C05477=1141.444,-110.919,-44.146,178.630,6.023,149.486
C05478=1141.449,-111.169,-44.137,178.627,6.022,149.487
C05479=1141.455,-111.418,-44.129,178.625,6.021,149.487
C05480=1141.460,-111.668,-44.120,178.624,6.021,149.488
C05481=1141.465,-111.918,-44.111,178.621,6.021,149.488
C05482=1141.470,-112.168,-44.102,178.620,6.021,149.489
C05483=1141.476,-112.417,-44.094,178.618,6.020,149.489
C05484=1141.481,-112.667,-44.085,178.616,6.020,149.490
C05485=1141.487,-112.917,-44.077,178.614,6.019,149.490
C05486=1141.492,-113.167,-44.068,178.612,6.019,149.491
C05487=1141.498,-113.416,-44.059,178.610,6.019,149.491
C05488=1141.503,-113.667,-44.051,178.607,6.018,149.492
C05489=1141.508,-113.916,-44.042,178.606,6.018,149.492
C05490=1141.513,-114.166,-44.033,178.604,6.018,149.493
C05491=1141.519,-114.415,-44.025,178.602,6.018,149.493
C05492=1141.524,-114.665,-44.016,178.600,6.017,149.494
C05493=1141.530,-114.916,-44.008,178.598,6.016,149.494
C05494=1141.535,-115.166,-43.999,178.596,6.016,149.495
C05495=1141.541,-115.415,-43.990,178.594,6.015,149.495
C05496=1141.546,-115.665,-43.981,178.592,6.015,149.496
C05497=1141.551,-115.915,-43.973,178.590,6.015,149.496
C05498=1141.557,-116.164,-43.964,178.588,6.015,149.497
C05499=1141.562,-116.414,-43.956,178.586,6.014,149.497
C05500=1141.567,-116.664,-43.947,178.585,6.014,149.498
C05501=1141.573,-116.914,-43.938,178.582,6.013,149.498
C05502=1141.579,-117.164,-43.930,178.580,6.013,149.499
C05503=1141.584,-117.413,-43.921,178.579,6.013,149.499
C05504=1141.589,-117.663,-43.912,178.576,6.012,149.500
C05505=1141.595,-117.913,-43.904,178.574,6.012,149.500
C05506=1141.600,-118.163,-43.895,178.572,6.012,149.501
C05507=1141.605,-118.412,-43.887,178.571,6.012,149.501
C05508=1141.611,-118.662,-43.879,178.568,6.011,149.502
C05509=1141.616,-118.912,-43.870,178.567,6.011,149.502
C05510=1141.621,-119.162,-43.862,178.565,6.010,149.503
C05511=1141.627,-119.412,-43.854,178.563,6.010,149.503
C05512=1141.632,-119.662,-43.845,178.561,6.009,149.504
C05513=1141.637,-119.911,-43.836,178.559,6.009,149.504
C05514=1141.644,-120.161,-43.828,178.557,6.009,149.505
C05515=1141.649,-120.411,-43.819,178.555,6.008,149.505
C05516=1141.653,-120.661,-43.811,178.553,6.008,149.506
C05517=1141.659,-120.910,-43.803,178.551,6.007,149.506
C05518=1141.664,-121.160,-43.794,178.549,6.007,149.507
C05519=1141.670,-121.411,-43.786,178.547,6.007,149.507
C05520=1141.676,-121.660,-43.777,178.546,6.007,149.508
C05521=1141.681,-121.910,-43.769,178.543,6.006,149.508
C05522=1141.686,-122.160,-43.760,178.542,6.006,149.509
C05523=1141.691,-122.409,-43.752,178.540,6.005,149.509
C05524=1141.697,-122.659,-43.744,178.538,6.005,149.510
C05525=1141.702,-122.909,-43.735,178.536,6.004,149.510
C05526=1141.708,-123.158,-43.727,178.534,6.004,149.511
C05527=1141.713,-123.409,-43.719,178.532,6.004,149.511
C05528=1141.719,-123.658,-43.710,178.530,6.003,149.512
C05529=1141.724,-123.908,-43.703,178.528,6.003,149.512
C05530=1141.729,-124.158,-43.694,178.526,6.002,149.513
C05531=1141.735,-124.408,-43.686,178.524,6.002,149.513
C05532=1141.740,-124.658,-43.677,178.522,6.002,149.514
C05533=1141.746,-124.908,-43.669,178.521,6.002,149.514
C05534=1141.751,-125.157,-43.661,178.518,6.001,149.515
C05535=1141.756,-125.407,-43.653,178.517,6.001,149.515
C05536=1141.762,-125.657,-43.644,178.515,6.000,149.516
C05537=1141.767,-125.907,-43.636,178.513,6.000,149.516
C05538=1141.772,-126.157,-43.628,178.511,6.000,149.517
C05539=1141.778,-126.406,-43.620,178.509,6.000,149.517
C05540=1141.783,-126.656,-43.611,178.507,5.999,149.518
C05541=1141.789,-126.906,-43.603,178.505,5.999,149.518
C05542=1141.794,-127.156,-43.594,178.503,5.998,149.519
C05543=1141.799,-127.405,-43.587,178.502,5.998,149.519
C05544=1141.805,-127.655,-43.578,178.499,5.997,149.519
C05545=1141.810,-127.906,-43.570,178.498,5.997,149.520
C05546=1141.816,-128.155,-43.561,178.496,5.997,149.520
C05547=1141.821,-128.405,-43.554,178.494,5.997,149.521
C05548=1141.400,-128.416,-43.597,178.490,6.000,149.523
C05549=1141.395,-128.166,-43.605,178.492,6.001,149.522
C05550=1141.389,-127.916,-43.613,178.494,6.001,149.522
C05551=1141.384,-127.667,-43.622,178.496,6.001,149.521
C05552=1141.378,-127.417,-43.629,178.498,6.001,149.521
C05553=1141.373,-127.167,-43.638,178.500,6.002,149.520
C05554=1141.367,-126.917,-43.646,178.502,6.002,149.520
C05555=1141.363,-126.668,-43.654,178.504,6.003,149.519
C05556=1141.357,-126.417,-43.663,178.505,6.003,149.519
C05557=1141.351,-126.168,-43.671,178.508,6.004,149.518
C05558=1141.346,-125.918,-43.679,178.509,6.004,149.518
C05559=1141.340,-125.668,-43.688,178.511,6.004,149.517
C05560=1141.335,-125.418,-43.695,178.513,6.004,149.517
C05561=1141.330,-125.168,-43.704,178.515,6.005,149.516
C05562=1141.324,-124.919,-43.712,178.517,6.005,149.516
C05563=1141.319,-124.669,-43.721,178.519,6.006,149.515
C05564=1141.314,-124.419,-43.728,178.521,6.006,149.515
C05565=1141.308,-124.169,-43.737,178.523,6.006,149.514
C05566=1141.303,-123.919,-43.745,178.524,6.006,149.514
C05567=1141.297,-123.670,-43.754,178.527,6.007,149.513
C05568=1141.292,-123.419,-43.762,178.528,6.007,149.513
C05569=1141.286,-123.170,-43.771,178.530,6.008,149.513
C05570=1141.281,-122.920,-43.778,178.533,6.009,149.512
C05571=1141.276,-122.670,-43.787,178.534,6.008,149.512
C05572=1141.270,-122.421,-43.796,178.536,6.009,149.511
C05573=1141.265,-122.171,-43.804,178.538,6.009,149.511
C05574=1141.260,-121.921,-43.813,178.540,6.010,149.510
C05575=1141.254,-121.671,-43.821,178.542,6.010,149.510
C05576=1141.249,-121.421,-43.829,178.544,6.011,149.509
C05577=1141.244,-121.172,-43.838,178.546,6.011,149.509
C05578=1141.238,-120.922,-43.846,178.548,6.011,149.508
C05579=1141.233,-120.672,-43.854,178.549,6.011,149.508
C05580=1141.228,-120.422,-43.863,178.552,6.012,149.507
C05581=1141.222,-120.172,-43.871,178.553,6.012,149.507
C05582=1141.216,-119.922,-43.880,178.555,6.013,149.506
C05583=1141.212,-119.672,-43.888,178.557,6.013,149.506
C05584=1141.206,-119.423,-43.896,178.559,6.013,149.505
C05585=1141.201,-119.173,-43.905,178.561,6.014,149.505
C05586=1141.195,-118.923,-43.913,178.563,6.014,149.504
C05587=1141.189,-118.674,-43.922,178.565,6.015,149.504
C05588=1141.184,-118.424,-43.931,178.567,6.014,149.503
C05589=1141.179,-118.173,-43.939,178.569,6.015,149.503
C05590=1141.173,-117.924,-43.947,178.571,6.015,149.502
C05591=1141.168,-117.674,-43.956,178.573,6.016,149.502
C05592=1141.163,-117.425,-43.965,178.575,6.016,149.501
C05593=1141.157,-117.175,-43.973,178.577,6.017,149.501
C05594=1141.152,-116.925,-43.981,178.579,6.017,149.500
C05595=1141.147,-116.675,-43.990,178.581,6.017,149.500
C05596=1141.141,-116.426,-43.998,178.583,6.018,149.499
C05597=1141.136,-116.176,-44.007,178.585,6.018,149.499
C05598=1141.131,-115.926,-44.016,178.587,6.019,149.498
C05599=1141.125,-115.676,-44.025,178.588,6.019,149.498
C05600=1141.119,-115.426,-44.033,178.591,6.019,149.497
C05601=1141.114,-115.176,-44.041,178.592,6.019,149.497
C05602=1141.109,-114.927,-44.050,178.594,6.020,149.496
C05603=1141.103,-114.677,-44.059,178.597,6.021,149.496
C05604=1141.098,-114.427,-44.067,178.598,6.021,149.495
C05605=1141.093,-114.177,-44.076,178.600,6.022,149.495
C05606=1141.088,-113.927,-44.085,178.602,6.022,149.494
C05607=1141.082,-113.678,-44.093,178.605,6.022,149.494
C05608=1141.077,-113.428,-44.102,178.606,6.022,149.493
C05609=1141.071,-113.178,-44.110,178.608,6.023,149.493
C05610=1141.066,-112.928,-44.119,178.611,6.023,149.492
C05611=1141.060,-112.679,-44.128,178.612,6.023,149.492
C05612=1141.055,-112.429,-44.137,178.614,6.024,149.491
C05613=1141.050,-112.179,-44.146,178.616,6.024,149.491
C05614=1141.045,-111.929,-44.155,178.618,6.025,149.490
C05615=1141.039,-111.679,-44.162,178.620,6.025,149.490
C05616=1141.033,-111.430,-44.171,178.622,6.025,149.489
C05617=1141.028,-111.180,-44.180,178.624,6.026,149.489
C05618=1141.023,-110.930,-44.189,178.626,6.026,149.488
C05619=1141.018,-110.680,-44.198,178.628,6.027,149.488
C05620=1141.012,-110.431,-44.207,178.630,6.027,149.487
C05621=1141.006,-110.181,-44.216,178.632,6.027,149.487
C05622=1141.001,-109.931,-44.225,178.634,6.027,149.486
C05623=1140.996,-109.680,-44.233,178.636,6.028,149.486
C05624=1140.990,-109.431,-44.242,178.638,6.029,149.485
C05625=1140.985,-109.181,-44.251,178.640,6.029,149.485
C05626=1140.980,-108.932,-44.259,178.642,6.029,149.484
C05627=1140.974,-108.682,-44.268,178.644,6.029,149.484
C05628=1140.969,-108.432,-44.277,178.646,6.030,149.483
C05629=1140.963,-108.183,-44.286,178.648,6.031,149.483
C05630=1140.958,-107.933,-44.295,178.650,6.031,149.482
C05631=1140.953,-107.683,-44.304,178.652,6.031,149.481
C05632=1140.948,-107.433,-44.312,178.654,6.031,149.481
C05633=1140.942,-107.183,-44.322,178.656,6.032,149.480
C05634=1140.937,-106.933,-44.331,178.658,6.033,149.480
C05635=1140.931,-106.684,-44.339,178.660,6.033,149.479
C05636=1140.926,-106.434,-44.348,178.662,6.033,149.479
C05637=1140.921,-106.184,-44.357,178.664,6.033,149.479
C05638=1140.916,-105.934,-44.366,178.666,6.034,149.478
C05639=1140.910,-105.685,-44.375,178.668,6.035,149.478
C05640=1140.905,-105.435,-44.384,178.670,6.035,149.477
C05641=1140.899,-105.185,-44.393,178.672,6.035,149.476
C05642=1140.894,-104.935,-44.402,178.674,6.035,149.476
C05643=1140.888,-104.686,-44.411,178.676,6.036,149.475
C05644=1140.883,-104.436,-44.420,178.678,6.037,149.475
C05645=1140.878,-104.186,-44.429,178.680,6.037,149.474
C05646=1140.873,-103.936,-44.437,178.682,6.037,149.474
C05647=1140.867,-103.686,-44.447,178.684,6.037,149.473
C05648=1140.862,-103.436,-44.456,178.686,6.038,149.473
C05649=1140.856,-103.165,-44.466,178.689,6.038,149.472
C05650=1140.850,-102.892,-44.475,178.691,6.039,149.472
C05651=1140.844,-102.620,-44.485,178.692,6.039,149.471
C05652=1140.839,-102.348,-44.495,178.695,6.039,149.471
C05653=1140.833,-102.098,-44.504,178.697,6.040,149.470
C05654=1140.828,-101.848,-44.513,178.699,6.040,149.470
C05655=1140.822,-101.598,-44.522,178.701,6.041,149.469
C05656=1140.817,-101.348,-44.531,178.703,6.042,149.469
C05657=1140.811,-101.099,-44.540,178.705,6.042,149.468
C05658=1140.807,-100.850,-44.549,178.707,6.042,149.468
C05659=1140.801,-100.600,-44.559,178.710,6.043,149.467
C05660=1140.796,-100.350,-44.568,178.711,6.043,149.466
C05661=1140.790,-100.100,-44.577,178.713,6.043,149.466
C05662=1140.785,-99.850,-44.585,178.715,6.043,149.465
C05663=1140.779,-99.600,-44.595,178.717,6.044,149.465
C05664=1140.774,-99.351,-44.605,178.719,6.045,149.464
C05665=1140.769,-99.101,-44.613,178.721,6.045,149.464
C05666=1140.763,-98.851,-44.623,178.724,6.045,149.463
C05667=1140.758,-98.601,-44.632,178.726,6.046,149.463
C05668=1140.753,-98.351,-44.641,178.728,6.046,149.462
C05669=1140.747,-98.102,-44.649,178.730,6.047,149.462
C05670=1140.742,-97.852,-44.660,178.732,6.047,149.461
C05671=1140.737,-97.602,-44.668,178.734,6.047,149.461
C05672=1140.731,-97.352,-44.677,178.736,6.048,149.460
C05673=1140.725,-97.102,-44.687,178.738,6.048,149.460
C05674=1140.721,-96.853,-44.696,178.740,6.049,149.459
C05675=1140.715,-96.603,-44.705,178.742,6.049,149.459
C05676=1140.710,-96.353,-44.715,178.744,6.049,149.458
C05677=1140.704,-96.103,-44.724,178.746,6.050,149.458
C05678=1140.699,-95.854,-44.733,178.748,6.051,149.457
C05679=1140.694,-95.604,-44.743,178.750,6.051,149.457
C05680=1140.688,-95.354,-44.752,178.752,6.051,149.456
C05681=1140.683,-95.104,-44.761,178.755,6.052,149.456
C05682=1140.678,-94.855,-44.771,178.756,6.052,149.455
C05683=1140.672,-94.605,-44.780,178.758,6.053,149.455
C05684=1140.667,-94.355,-44.789,178.761,6.053,149.454
C05685=1140.662,-94.105,-44.799,178.762,6.053,149.454
C05686=1140.657,-93.855,-44.808,178.765,6.054,149.453
C05687=1140.651,-93.606,-44.817,178.767,6.054,149.452
C05688=1140.646,-93.356,-44.827,178.769,6.054,149.452
C05689=1140.641,-93.106,-44.836,178.771,6.055,149.451
C05690=1140.635,-92.856,-44.845,178.773,6.056,149.451
C05691=1140.630,-92.607,-44.855,178.775,6.056,149.450
C05692=1140.625,-92.357,-44.864,178.777,6.056,149.450
C05693=1140.619,-92.107,-44.873,178.780,6.057,149.449
C05694=1140.614,-91.858,-44.883,178.781,6.057,149.449
C05695=1140.608,-91.607,-44.892,178.783,6.058,149.448
C05696=1140.603,-91.358,-44.901,178.786,6.058,149.448
C05697=1140.598,-91.108,-44.911,178.787,6.058,149.447
C05698=1140.592,-90.858,-44.920,178.790,6.059,149.447
C05699=1140.587,-90.609,-44.930,178.792,6.060,149.446
C05700=1140.581,-90.359,-44.939,178.794,6.060,149.446
C05701=1140.576,-90.109,-44.948,178.796,6.060,149.445
C05702=1140.571,-89.859,-44.959,178.798,6.061,149.445
C05703=1140.565,-89.610,-44.967,178.800,6.061,149.444
C05704=1140.560,-89.360,-44.978,178.802,6.061,149.443
C05705=1140.555,-89.110,-44.987,178.804,6.062,149.443
C05706=1140.550,-88.860,-44.997,178.806,6.062,149.443
C05707=1140.544,-88.610,-45.006,178.808,6.063,149.442
C05708=1140.540,-88.361,-45.016,178.810,6.064,149.442
C05709=1140.534,-88.111,-45.025,178.813,6.064,149.441
C05710=1140.529,-87.861,-45.034,178.815,6.064,149.440
C05711=1140.523,-87.611,-45.044,178.817,6.065,149.440
C05712=1140.518,-87.361,-45.053,178.819,6.065,149.439
C05713=1140.512,-87.112,-45.063,178.821,6.065,149.439
C05714=1140.507,-86.862,-45.072,178.823,6.066,149.438
C05715=1140.501,-86.612,-45.082,178.826,6.067,149.438
C05716=1140.496,-86.363,-45.091,178.827,6.067,149.437
C05717=1140.491,-86.113,-45.102,178.829,6.067,149.437
C05718=1140.486,-85.863,-45.112,178.831,6.068,149.436
C05719=1140.480,-85.613,-45.121,178.834,6.068,149.436
C05720=1140.476,-85.364,-45.131,178.836,6.068,149.435
C05721=1140.470,-85.114,-45.140,178.838,6.069,149.435
C05722=1140.465,-84.864,-45.150,178.840,6.070,149.434
C05723=1140.459,-84.614,-45.159,178.842,6.070,149.434
C05724=1140.453,-84.365,-45.169,178.844,6.070,149.433
C05725=1140.448,-84.115,-45.178,178.847,6.071,149.432
C05726=1140.443,-83.865,-45.189,178.849,6.072,149.432
C05727=1140.438,-83.615,-45.199,178.850,6.072,149.431
C05728=1140.432,-83.365,-45.208,178.853,6.072,149.431
C05729=1140.428,-83.116,-45.218,178.855,6.073,149.430
C05730=1140.422,-82.866,-45.227,178.857,6.073,149.430
C05731=1140.416,-82.616,-45.237,178.859,6.074,149.429
C05732=1140.411,-82.367,-45.247,178.861,6.074,149.429
C05733=1140.406,-82.116,-45.257,178.863,6.075,149.428
C05734=1140.401,-81.867,-45.266,178.866,6.075,149.428
C05735=1140.395,-81.617,-45.277,178.868,6.075,149.427
C05736=1140.390,-81.367,-45.286,178.870,6.076,149.427
C05737=1140.385,-81.118,-45.296,178.871,6.076,149.426
C05738=1140.379,-80.868,-45.306,178.874,6.077,149.425
C05739=1140.375,-80.618,-45.315,178.876,6.077,149.425
C05740=1140.369,-80.368,-45.325,178.879,6.078,149.424
C05741=1140.363,-80.119,-45.336,178.880,6.078,149.424
C05742=1140.358,-79.869,-45.345,178.882,6.079,149.424
C05743=1140.353,-79.619,-45.355,178.885,6.079,149.423
C05744=1140.347,-79.370,-45.365,178.887,6.080,149.422
C05745=1140.343,-79.120,-45.375,178.889,6.080,149.422
C05746=1140.337,-78.870,-45.384,178.891,6.081,149.421
C05747=1140.331,-78.620,-45.395,178.894,6.081,149.421
C05748=1140.326,-78.371,-45.404,178.896,6.082,149.420
C05749=1140.320,-78.121,-45.414,178.897,6.082,149.420
C05750=1140.315,-77.871,-45.424,178.900,6.083,149.419
C05751=1140.310,-77.621,-45.435,178.902,6.083,149.419
C05752=1140.305,-77.372,-45.444,178.905,6.084,149.418
C05753=1140.299,-77.100,-45.455,178.906,6.084,149.418
C05754=1140.293,-76.829,-45.466,178.909,6.084,149.417
C05755=1140.287,-76.557,-45.477,178.911,6.085,149.416
C05756=1140.282,-76.285,-45.487,178.913,6.086,149.416
C05757=1140.276,-76.036,-45.498,178.916,6.086,149.415
C05758=1140.271,-75.787,-45.507,178.918,6.087,149.415
C05759=1140.266,-75.536,-45.518,178.920,6.087,149.414
C05760=1140.260,-75.287,-45.528,178.922,6.087,149.414
C05761=1140.255,-75.037,-45.537,178.925,6.088,149.413
C05762=1140.250,-74.787,-45.547,178.927,6.089,149.412
C05763=1140.244,-74.538,-45.557,178.928,6.088,149.412
C05764=1140.239,-74.288,-45.568,178.930,6.089,149.412
C05765=1140.234,-74.038,-45.578,178.933,6.090,149.411
C05766=1140.228,-73.789,-45.588,178.935,6.090,149.410
C05767=1140.223,-73.538,-45.597,178.938,6.091,149.410
C05768=1140.218,-73.288,-45.608,178.939,6.091,149.409
C05769=1140.212,-73.039,-45.618,178.942,6.092,149.409
C05770=1140.207,-72.789,-45.628,178.944,6.092,149.408
C05771=1140.202,-72.539,-45.638,178.946,6.093,149.408
C05772=1140.197,-72.290,-45.648,178.948,6.093,149.407
C05773=1140.191,-72.040,-45.659,178.950,6.093,149.407
C05774=1140.185,-71.791,-45.669,178.953,6.094,149.406
C05775=1140.181,-71.541,-45.679,178.955,6.095,149.406
C05776=1140.175,-71.291,-45.689,178.956,6.095,149.405
C05777=1140.170,-71.042,-45.699,178.959,6.095,149.404
C05778=1140.165,-70.792,-45.710,178.961,6.096,149.404
C05779=1140.159,-70.542,-45.720,178.963,6.097,149.403
C05780=1140.154,-70.292,-45.729,178.966,6.098,149.403
C05781=1140.149,-70.042,-45.740,178.968,6.097,149.402
C05782=1140.143,-69.792,-45.750,178.970,6.098,149.402
C05783=1140.138,-69.543,-45.760,178.972,6.099,149.401
C05784=1140.133,-69.293,-45.770,178.974,6.099,149.401
C05785=1140.127,-69.043,-45.781,178.977,6.100,149.400
C05786=1140.122,-68.794,-45.791,178.979,6.100,149.400
C05787=1140.117,-68.543,-45.801,178.981,6.101,149.399
C05788=1140.111,-68.294,-45.812,178.983,6.101,149.399
C05789=1140.106,-68.045,-45.822,178.986,6.102,149.398
C05790=1140.101,-67.795,-45.833,178.988,6.102,149.397
C05791=1140.095,-67.545,-45.843,178.989,6.102,149.397
C05792=1140.091,-67.296,-45.853,178.992,6.103,149.396
C05793=1140.086,-67.046,-45.863,178.994,6.104,149.396
C05794=1140.080,-66.796,-45.874,178.996,6.104,149.395
C05795=1140.074,-66.546,-45.884,178.999,6.105,149.395
C05796=1140.069,-66.296,-45.894,179.001,6.105,149.394
C05797=1140.064,-66.047,-45.905,179.003,6.106,149.394
C05798=1140.059,-65.796,-45.915,179.005,6.106,149.393
C05799=1140.053,-65.547,-45.925,179.007,6.107,149.393
C05800=1140.048,-65.297,-45.936,179.010,6.107,149.392
C05801=1140.043,-65.047,-45.946,179.012,6.107,149.391
C05802=1140.037,-64.798,-45.957,179.014,6.108,149.391
C05803=1140.032,-64.548,-45.968,179.016,6.109,149.390
C05804=1140.027,-64.298,-45.978,179.019,6.109,149.390
C05805=1140.021,-64.049,-45.988,179.021,6.110,149.389
C05806=1140.016,-63.799,-45.999,179.023,6.111,149.389
C05807=1140.010,-63.549,-46.009,179.025,6.110,149.388
C05808=1140.006,-63.299,-46.020,179.027,6.111,149.388
C05809=1140.000,-63.050,-46.030,179.029,6.112,149.387
C05810=1139.995,-62.800,-46.041,179.032,6.113,149.387
C05811=1139.990,-62.550,-46.051,179.034,6.113,149.386
C05812=1139.984,-62.301,-46.061,179.036,6.113,149.385
C05813=1139.979,-62.051,-46.073,179.038,6.114,149.385
C05814=1139.974,-61.801,-46.083,179.041,6.114,149.384
C05815=1139.969,-61.551,-46.093,179.043,6.115,149.384
C05816=1139.963,-61.302,-46.104,179.045,6.116,149.383
C05817=1139.958,-61.051,-46.114,179.047,6.117,149.383
C05818=1139.953,-60.802,-46.125,179.049,6.116,149.382
C05819=1139.947,-60.553,-46.135,179.052,6.117,149.382
C05820=1139.942,-60.303,-46.146,179.054,6.118,149.381
C05821=1139.937,-60.053,-46.156,179.056,6.118,149.380
C05822=1139.932,-59.803,-46.167,179.059,6.119,149.380
C05823=1139.926,-59.554,-46.178,179.061,6.120,149.380
C05824=1139.921,-59.304,-46.188,179.063,6.120,149.379
C05825=1139.916,-59.055,-46.199,179.065,6.120,149.378
C05826=1139.911,-58.805,-46.210,179.067,6.121,149.378
C05827=1139.905,-58.555,-46.220,179.069,6.122,149.377
C05828=1139.901,-58.305,-46.231,179.072,6.122,149.377
C05829=1139.895,-58.056,-46.241,179.074,6.123,149.376
C05830=1139.890,-57.806,-46.252,179.077,6.123,149.376
C05831=1139.885,-57.557,-46.263,179.079,6.124,149.375
C05832=1139.879,-57.306,-46.274,179.081,6.124,149.375
C05833=1139.874,-57.057,-46.284,179.083,6.125,149.374
C05834=1139.869,-56.807,-46.296,179.085,6.125,149.374
C05835=1139.863,-56.557,-46.306,179.088,6.126,149.373
C05836=1139.858,-56.307,-46.316,179.090,6.127,149.372
C05837=1139.853,-56.058,-46.327,179.092,6.127,149.372
C05838=1139.848,-55.808,-46.338,179.095,6.128,149.371
C05839=1139.843,-55.559,-46.349,179.096,6.128,149.371
C05840=1139.837,-55.308,-46.360,179.099,6.128,149.370
C05841=1139.831,-55.059,-46.370,179.101,6.129,149.370
C05842=1139.827,-54.809,-46.381,179.104,6.130,149.369
C05843=1139.822,-54.559,-46.392,179.106,6.130,149.369
C05844=1139.816,-54.310,-46.403,179.108,6.131,149.368
C05845=1139.811,-54.060,-46.414,179.111,6.132,149.367
C05846=1139.805,-53.811,-46.425,179.113,6.132,149.367
C05847=1139.800,-53.560,-46.436,179.114,6.132,149.366
C05848=1139.795,-53.311,-46.447,179.117,6.133,149.366
C05849=1139.790,-53.061,-46.457,179.119,6.133,149.365
C05850=1139.784,-52.812,-46.467,179.121,6.134,149.365
C05851=1139.779,-52.562,-46.479,179.124,6.135,149.364
C05852=1139.774,-52.311,-46.490,179.126,6.135,149.364
C05853=1139.769,-52.063,-46.501,179.128,6.136,149.363
C05854=1139.764,-51.812,-46.511,179.131,6.137,149.363
C05855=1139.758,-51.563,-46.523,179.133,6.137,149.362
C05856=1139.753,-51.313,-46.534,179.135,6.137,149.361
C05857=1139.747,-51.042,-46.546,179.138,6.138,149.361
C05858=1139.742,-50.772,-46.557,179.140,6.138,149.360
C05859=1139.736,-50.501,-46.569,179.143,6.140,149.360
C05860=1139.730,-50.230,-46.581,179.145,6.140,149.359
C05861=1139.725,-49.981,-46.592,179.147,6.140,149.359
C05862=1139.720,-49.731,-46.603,179.149,6.141,149.358
C05863=1139.714,-49.482,-46.614,179.152,6.142,149.357
C05864=1139.709,-49.231,-46.625,179.154,6.142,149.357
C05865=1139.704,-48.982,-46.636,179.157,6.143,149.356
C05866=1139.698,-48.732,-46.648,179.159,6.144,149.356
C05867=1139.693,-48.482,-46.658,179.161,6.144,149.355
C05868=1139.688,-48.233,-46.669,179.164,6.145,149.355
C05869=1139.682,-47.983,-46.681,179.166,6.145,149.354
C05870=1139.678,-47.733,-46.692,179.168,6.146,149.354
C05871=1139.672,-47.484,-46.703,179.171,6.147,149.353
C05872=1139.667,-47.234,-46.713,179.172,6.147,149.352
C05873=1139.662,-46.984,-46.725,179.174,6.147,149.352
C05874=1139.657,-46.735,-46.736,179.177,6.148,149.352
C05875=1139.651,-46.484,-46.747,179.179,6.149,149.351
C05876=1139.646,-46.235,-46.759,179.181,6.149,149.350
C05877=1139.641,-45.986,-46.770,179.184,6.150,149.350
C05878=1139.635,-45.735,-46.781,179.186,6.151,149.349
C05879=1139.630,-45.486,-46.792,179.188,6.151,149.349
C05880=1139.625,-45.237,-46.803,179.191,6.152,149.348
C05881=1139.620,-44.987,-46.815,179.193,6.152,149.347
C05882=1139.615,-44.737,-46.825,179.196,6.153,149.347
C05883=1139.609,-44.488,-46.836,179.198,6.154,149.347
C05884=1139.604,-44.238,-46.848,179.200,6.154,149.346
C05885=1139.599,-43.988,-46.859,179.203,6.155,149.345
C05886=1139.593,-43.738,-46.870,179.204,6.155,149.345
C05887=1139.588,-43.489,-46.882,179.207,6.156,149.344
C05888=1139.583,-43.239,-46.893,179.209,6.156,149.344
C05889=1139.578,-42.989,-46.905,179.211,6.157,149.343
C05890=1139.573,-42.740,-46.915,179.214,6.158,149.343
C05891=1139.567,-42.490,-46.927,179.216,6.158,149.342
C05892=1139.562,-42.240,-46.938,179.218,6.159,149.342
C05893=1139.556,-41.991,-46.950,179.221,6.160,149.341
C05894=1139.552,-41.741,-46.961,179.223,6.160,149.340
C05895=1139.546,-41.491,-46.972,179.225,6.161,149.340
C05896=1139.541,-41.241,-46.983,179.228,6.161,149.339
C05897=1139.535,-40.992,-46.995,179.230,6.162,149.339
C05898=1139.531,-40.742,-47.006,179.232,6.163,149.338
C05899=1139.526,-40.493,-47.017,179.235,6.163,149.338
C05900=1139.520,-40.243,-47.029,179.237,6.164,149.337
C05901=1139.515,-39.994,-47.040,179.239,6.165,149.337
C05902=1139.509,-39.743,-47.051,179.242,6.165,149.336
C05903=1139.505,-39.493,-47.063,179.244,6.166,149.335
C05904=1139.499,-39.244,-47.075,179.246,6.167,149.335
C05905=1139.493,-38.994,-47.086,179.249,6.167,149.334
C05906=1139.489,-38.745,-47.097,179.251,6.167,149.334
C05907=1139.483,-38.495,-47.109,179.253,6.168,149.333
C05908=1139.478,-38.245,-47.121,179.256,6.169,149.333
C05909=1139.473,-37.995,-47.133,179.258,6.169,149.332
C05910=1139.468,-37.746,-47.143,179.260,6.170,149.332
C05911=1139.462,-37.496,-47.155,179.263,6.170,149.331
C05912=1139.458,-37.247,-47.167,179.265,6.171,149.330
C05913=1139.452,-36.997,-47.178,179.267,6.172,149.330
C05914=1139.447,-36.747,-47.190,179.270,6.172,149.329
C05915=1139.441,-36.498,-47.201,179.272,6.173,149.329
C05916=1139.436,-36.248,-47.213,179.274,6.174,149.328
C05917=1139.431,-35.998,-47.224,179.277,6.174,149.328
C05918=1139.426,-35.748,-47.236,179.279,6.175,149.327
C05919=1139.421,-35.499,-47.248,179.281,6.176,149.326
C05920=1139.415,-35.250,-47.259,179.284,6.176,149.326
C05921=1139.410,-35.000,-47.271,179.286,6.177,149.326
C05922=1139.405,-34.750,-47.282,179.289,6.178,149.325
C05923=1139.400,-34.500,-47.294,179.291,6.178,149.324
C05924=1139.395,-34.250,-47.306,179.293,6.179,149.324
C05925=1139.390,-34.000,-47.317,179.296,6.180,149.323
C05926=1139.383,-33.751,-47.329,179.298,6.180,149.323
C05927=1139.379,-33.502,-47.340,179.300,6.181,149.322
C05928=1139.373,-33.252,-47.352,179.303,6.181,149.322
C05929=1139.368,-33.002,-47.364,179.305,6.182,149.321
C05930=1139.363,-32.752,-47.375,179.307,6.183,149.321
C05931=1139.358,-32.502,-47.387,179.310,6.183,149.320
C05932=1139.353,-32.253,-47.400,179.312,6.184,149.319
C05933=1139.347,-32.004,-47.411,179.314,6.185,149.319
C05934=1139.342,-31.754,-47.423,179.317,6.185,149.318
C05935=1139.337,-31.504,-47.434,179.319,6.186,149.318
C05936=1139.332,-31.254,-47.446,179.321,6.187,149.317
C05937=1139.326,-31.004,-47.458,179.324,6.187,149.317
C05938=1139.321,-30.755,-47.470,179.326,6.188,149.316
C05939=1139.317,-30.506,-47.482,179.328,6.189,149.316
C05940=1139.311,-30.256,-47.493,179.331,6.189,149.315
C05941=1139.306,-30.006,-47.505,179.333,6.190,149.314
C05942=1139.300,-29.756,-47.517,179.336,6.191,149.314
C05943=1139.295,-29.507,-47.528,179.338,6.191,149.313
C05944=1139.290,-29.258,-47.541,179.340,6.192,149.313
C05945=1139.284,-29.008,-47.553,179.343,6.193,149.312
C05946=1139.280,-28.758,-47.564,179.345,6.193,149.312
C05947=1139.274,-28.508,-47.576,179.347,6.194,149.311
C05948=1139.269,-28.259,-47.588,179.350,6.195,149.310
C05949=1139.264,-28.009,-47.600,179.352,6.195,149.310
C05950=1139.259,-27.759,-47.612,179.354,6.196,149.310
C05951=1139.254,-27.509,-47.623,179.357,6.197,149.309
C05952=1139.249,-27.260,-47.636,179.359,6.198,149.308
C05953=1139.243,-27.010,-47.648,179.362,6.199,149.308
C05954=1139.238,-26.760,-47.660,179.364,6.199,149.307
C05955=1139.233,-26.510,-47.671,179.366,6.200,149.307
C05956=1139.228,-26.261,-47.684,179.369,6.200,149.306
C05957=1139.222,-26.011,-47.696,179.371,6.201,149.306
C05958=1139.217,-25.761,-47.707,179.374,6.202,149.305
C05959=1139.212,-25.512,-47.720,179.376,6.202,149.304
C05960=1139.207,-25.262,-47.731,179.378,6.203,149.304
C05961=1139.201,-24.992,-47.745,179.381,6.204,149.303
C05962=1139.195,-24.722,-47.758,179.383,6.204,149.303
C05963=1139.190,-24.452,-47.770,179.386,6.206,149.302
C05964=1139.184,-24.183,-47.784,179.389,6.206,149.302
C05965=1139.179,-23.933,-47.796,179.391,6.207,149.301
C05966=1139.173,-23.683,-47.808,179.394,6.208,149.300
C05967=1139.168,-23.433,-47.820,179.396,6.208,149.300
C05968=1139.163,-23.183,-47.832,179.398,6.209,149.299
C05969=1139.159,-22.934,-47.844,179.401,6.210,149.299
C05970=1139.153,-22.684,-47.856,179.403,6.210,149.298
C05971=1139.148,-22.435,-47.868,179.405,6.211,149.298
C05972=1139.143,-22.185,-47.880,179.408,6.212,149.297
C05973=1139.137,-21.935,-47.892,179.410,6.212,149.297
C05974=1139.132,-21.686,-47.905,179.412,6.213,149.296
C05975=1139.127,-21.436,-47.917,179.415,6.214,149.295
C05976=1139.121,-21.187,-47.929,179.418,6.215,149.295
C05977=1139.117,-20.936,-47.942,179.420,6.216,149.294
C05978=1139.111,-20.687,-47.954,179.422,6.216,149.294
C05979=1139.106,-20.437,-47.966,179.425,6.217,149.293
C05980=1139.101,-20.187,-47.979,179.427,6.218,149.293
C05981=1139.096,-19.938,-47.991,179.429,6.218,149.292
C05982=1139.091,-19.689,-48.003,179.432,6.219,149.291
C05983=1139.086,-19.439,-48.015,179.434,6.220,149.291
C05984=1139.081,-19.189,-48.027,179.436,6.220,149.291
C05985=1139.075,-18.939,-48.039,179.439,6.221,149.290
C05986=1139.070,-18.690,-48.052,179.441,6.222,149.289
C05987=1139.065,-18.441,-48.064,179.444,6.222,149.289
C05988=1139.059,-18.191,-48.076,179.447,6.224,149.288
C05989=1139.054,-17.941,-48.089,179.449,6.224,149.288
C05990=1139.049,-17.692,-48.101,179.451,6.225,149.287
C05991=1139.044,-17.442,-48.114,179.454,6.226,149.287
C05992=1139.039,-17.192,-48.125,179.456,6.226,149.286
C05993=1139.034,-16.942,-48.138,179.458,6.227,149.285
C05994=1139.029,-16.693,-48.151,179.461,6.228,149.285
C05995=1139.023,-16.443,-48.163,179.463,6.228,149.284
C05996=1139.018,-16.194,-48.175,179.465,6.229,149.284
C05997=1139.013,-15.944,-48.188,179.468,6.230,149.283
C05998=1139.007,-15.694,-48.200,179.471,6.231,149.283
C05999=1139.002,-15.444,-48.213,179.473,6.232,149.282
C06000=1138.997,-15.195,-48.226,179.475,6.232,149.282
C06001=1138.992,-14.945,-48.238,179.478,6.233,149.281
C06002=1138.987,-14.696,-48.250,179.480,6.234,149.281
C06003=1138.982,-14.446,-48.263,179.482,6.234,149.280
C06004=1138.976,-14.196,-48.275,179.485,6.235,149.279
C06005=1138.971,-13.947,-48.287,179.487,6.236,149.279
C06006=1138.966,-13.697,-48.300,179.490,6.236,149.278
C06007=1138.961,-13.448,-48.313,179.493,6.238,149.278
C06008=1138.956,-13.198,-48.325,179.495,6.238,149.277
C06009=1138.951,-12.948,-48.337,179.497,6.239,149.277
C06010=1138.945,-12.699,-48.351,179.500,6.240,149.276
C06011=1138.940,-12.449,-48.364,179.502,6.240,149.276
C06012=1138.935,-12.199,-48.375,179.504,6.241,149.275
C06013=1138.930,-11.949,-48.388,179.507,6.242,149.274
C06014=1138.925,-11.700,-48.401,179.509,6.242,149.274
C06015=1138.920,-11.451,-48.413,179.512,6.244,149.273
C06016=1138.914,-11.202,-48.426,179.514,6.244,149.273
C06017=1138.910,-10.951,-48.438,179.517,6.245,149.272
C06018=1138.904,-10.701,-48.451,179.519,6.246,149.272
C06019=1138.899,-10.452,-48.464,179.521,6.246,149.271
C06020=1138.894,-10.203,-48.476,179.524,6.247,149.271
C06021=1138.889,-9.953,-48.489,179.526,6.248,149.270
C06022=1138.884,-9.703,-48.502,179.529,6.249,149.270
C06023=1138.878,-9.453,-48.515,179.532,6.250,149.269
C06024=1138.873,-9.204,-48.527,179.534,6.251,149.268
C06025=1138.868,-8.954,-48.540,179.536,6.251,149.268
C06026=1138.863,-8.704,-48.553,179.539,6.252,149.267
C06027=1138.858,-8.455,-48.565,179.541,6.253,149.267
C06028=1138.852,-8.205,-48.578,179.543,6.253,149.266
C06029=1138.847,-7.955,-48.591,179.546,6.255,149.266
C06030=1138.842,-7.706,-48.604,179.548,6.255,149.265
C06031=1138.837,-7.457,-48.617,179.551,6.256,149.264
C06032=1138.831,-7.207,-48.630,179.553,6.257,149.264
C06033=1138.827,-6.957,-48.643,179.556,6.257,149.263
C06034=1138.822,-6.708,-48.655,179.558,6.258,149.263
C06035=1138.817,-6.458,-48.668,179.561,6.259,149.262
C06036=1138.811,-6.209,-48.681,179.563,6.260,149.262
C06037=1138.806,-5.959,-48.694,179.566,6.261,149.261
C06038=1138.801,-5.710,-48.707,179.568,6.261,149.261
C06039=1138.796,-5.460,-48.719,179.570,6.262,149.260
C06040=1138.791,-5.210,-48.733,179.573,6.263,149.260
C06041=1138.786,-4.961,-48.746,179.576,6.264,149.259
C06042=1138.780,-4.711,-48.758,179.578,6.265,149.258
C06043=1138.775,-4.461,-48.772,179.580,6.265,149.258
C06044=1138.770,-4.212,-48.784,179.583,6.266,149.257
C06045=1138.765,-3.962,-48.797,179.585,6.267,149.257
C06046=1138.760,-3.712,-48.810,179.588,6.268,149.256
C06047=1138.755,-3.463,-48.823,179.591,6.269,149.256
C06048=1138.749,-3.213,-48.836,179.593,6.269,149.255
C06049=1138.744,-2.963,-48.849,179.595,6.270,149.254
C06050=1138.739,-2.714,-48.862,179.598,6.271,149.254
C06051=1138.734,-2.464,-48.874,179.600,6.272,149.254
C06052=1138.729,-2.214,-48.888,179.603,6.273,149.253
C06053=1138.724,-1.965,-48.901,179.605,6.274,149.252
C06054=1138.718,-1.716,-48.915,179.607,6.274,149.252
C06055=1138.713,-1.466,-48.927,179.610,6.275,149.251
C06056=1138.708,-1.216,-48.940,179.613,6.276,149.251
C06057=1138.702,-0.967,-48.953,179.615,6.277,149.250
C06058=1138.698,-0.717,-48.966,179.618,6.278,149.250
C06059=1138.692,-0.467,-48.979,179.620,6.278,149.249
C06060=1138.687,-0.218,-48.993,179.622,6.279,149.248
C06061=1138.683,0.032,-49.006,179.625,6.280,149.248
C06062=1138.677,0.281,-49.019,179.627,6.281,149.248
C06063=1138.672,0.531,-49.032,179.630,6.282,149.247
C06064=1138.666,0.781,-49.045,179.632,6.282,149.246
C06065=1138.662,1.050,-49.059,179.635,6.284,149.246
C06066=1138.655,1.319,-49.073,179.638,6.284,149.245
C06067=1138.650,1.589,-49.088,179.640,6.285,149.245
C06068=1138.645,1.858,-49.102,179.643,6.287,149.244
C06069=1138.639,2.108,-49.115,179.646,6.287,149.243
C06070=1138.635,2.358,-49.128,179.648,6.288,149.243
C06071=1138.629,2.607,-49.142,179.651,6.288,149.242
C06072=1138.625,2.857,-49.155,179.653,6.290,149.242
C06073=1138.619,3.107,-49.168,179.656,6.291,149.241
C06074=1138.614,3.355,-49.182,179.658,6.291,149.241
C06075=1138.609,3.606,-49.195,179.660,6.292,149.240
C06076=1138.603,3.855,-49.208,179.663,6.293,149.240
C06077=1138.599,4.105,-49.222,179.666,6.294,149.239
C06078=1138.593,4.354,-49.235,179.668,6.295,149.239
C06079=1138.588,4.605,-49.248,179.671,6.295,149.238
C06080=1138.583,4.853,-49.262,179.673,6.297,149.237
C06081=1138.578,5.104,-49.275,179.676,6.297,149.237
C06082=1138.572,5.353,-49.288,179.678,6.298,149.236
C06083=1138.568,5.603,-49.302,179.680,6.299,149.236
C06084=1138.562,5.852,-49.315,179.683,6.300,149.235
C06085=1138.558,6.102,-49.329,179.686,6.301,149.235
C06086=1138.552,6.351,-49.342,179.688,6.302,149.234
C06087=1138.548,6.601,-49.355,179.691,6.302,149.233
C06088=1138.542,6.850,-49.369,179.693,6.304,149.233
C06089=1138.537,7.101,-49.382,179.696,6.304,149.233
C06090=1138.532,7.349,-49.396,179.698,6.305,149.232
C06091=1138.527,7.600,-49.409,179.700,6.306,149.231
C06092=1138.522,7.848,-49.423,179.703,6.307,149.231
C06093=1138.517,8.099,-49.436,179.706,6.308,149.230
C06094=1138.511,8.348,-49.450,179.708,6.308,149.230
C06095=1138.506,8.598,-49.463,179.711,6.309,149.229
C06096=1138.501,8.847,-49.477,179.713,6.311,149.229
C06097=1138.496,9.097,-49.491,179.716,6.311,149.228
C06098=1138.491,9.346,-49.504,179.718,6.312,149.227
C06099=1138.486,9.596,-49.517,179.720,6.313,149.227
C06100=1138.480,9.845,-49.531,179.723,6.314,149.227
C06101=1138.475,10.095,-49.544,179.726,6.315,149.226
C06102=1138.470,10.344,-49.558,179.728,6.315,149.225
C06103=1138.465,10.594,-49.572,179.731,6.317,149.225
C06104=1138.460,10.844,-49.585,179.733,6.317,149.224
C06105=1138.455,11.093,-49.599,179.736,6.318,149.224
C06106=1138.450,11.343,-49.613,179.738,6.319,149.223
C06107=1138.445,11.592,-49.626,179.741,6.320,149.223
C06108=1138.440,11.842,-49.640,179.743,6.321,149.222
C06109=1138.434,12.091,-49.654,179.746,6.322,149.222
C06110=1138.429,12.341,-49.668,179.749,6.323,149.221
C06111=1138.425,12.591,-49.681,179.751,6.324,149.221
C06112=1138.419,12.840,-49.695,179.753,6.324,149.220
C06113=1138.414,13.090,-49.708,179.756,6.325,149.219
C06114=1138.408,13.339,-49.722,179.759,6.326,149.219
C06115=1138.404,13.589,-49.736,179.761,6.327,149.218
C06116=1138.399,13.839,-49.750,179.763,6.328,149.218
C06117=1138.393,14.088,-49.764,179.767,6.329,149.217
C06118=1138.388,14.338,-49.778,179.769,6.330,149.217
C06119=1138.384,14.587,-49.791,179.771,6.331,149.216
C06120=1138.378,14.837,-49.805,179.774,6.332,149.216
C06121=1138.373,15.086,-49.819,179.776,6.333,149.215
C06122=1138.368,15.335,-49.833,179.779,6.333,149.214
C06123=1138.362,15.586,-49.846,179.781,6.334,149.214
C06124=1138.358,15.835,-49.860,179.784,6.336,149.214
C06125=1138.353,16.084,-49.874,179.787,6.336,149.213
C06126=1138.348,16.334,-49.888,179.789,6.337,149.212
C06127=1138.342,16.584,-49.902,179.791,6.339,149.212
C06128=1138.337,16.833,-49.916,179.794,6.339,149.211
C06129=1138.332,17.083,-49.930,179.796,6.340,149.211
C06130=1138.328,17.332,-49.944,179.799,6.342,149.210
C06131=1138.322,17.581,-49.958,179.802,6.342,149.210
C06132=1138.317,17.832,-49.971,179.804,6.343,149.209
C06133=1138.312,18.081,-49.985,179.807,6.344,149.208
C06134=1138.306,18.330,-49.999,179.809,6.345,149.208
C06135=1138.301,18.580,-50.014,179.811,6.346,149.208
C06136=1138.296,18.830,-50.028,179.815,6.347,149.207
C06137=1138.291,19.080,-50.042,179.817,6.348,149.206
C06138=1138.286,19.329,-50.056,179.819,6.349,149.206
C06139=1138.281,19.579,-50.069,179.822,6.350,149.205
C06140=1138.276,19.828,-50.083,179.824,6.351,149.205
C06141=1138.271,20.077,-50.097,179.827,6.351,149.204
C06142=1138.266,20.327,-50.112,179.830,6.353,149.204
C06143=1138.261,20.577,-50.126,179.832,6.354,149.203
C06144=1138.256,20.826,-50.140,179.835,6.354,149.203
C06145=1138.250,21.075,-50.154,179.838,6.356,149.202
C06146=1138.245,21.325,-50.168,179.840,6.356,149.202
C06147=1138.240,21.575,-50.183,179.843,6.358,149.201
C06148=1138.236,21.825,-50.197,179.845,6.358,149.200
C06149=1138.230,22.074,-50.211,179.847,6.359,149.200
C06150=1138.225,22.323,-50.225,179.851,6.360,149.199
C06151=1138.220,22.573,-50.239,179.853,6.361,149.199
C06152=1138.215,22.823,-50.254,179.855,6.362,149.198
C06153=1138.210,23.072,-50.268,179.858,6.363,149.198
C06154=1138.205,23.321,-50.282,179.860,6.364,149.197
C06155=1138.200,23.571,-50.296,179.863,6.365,149.197
C06156=1138.195,23.821,-50.310,179.866,6.366,149.196
C06157=1138.190,24.071,-50.325,179.868,6.367,149.196
C06158=1138.184,24.320,-50.339,179.871,6.368,149.195
C06159=1138.179,24.569,-50.353,179.873,6.369,149.195
C06160=1138.174,24.819,-50.367,179.875,6.370,149.194
C06161=1138.169,25.069,-50.381,179.879,6.371,149.193
C06162=1138.164,25.318,-50.396,179.881,6.372,149.193
C06163=1138.159,25.567,-50.410,179.883,6.373,149.193
C06164=1138.154,25.816,-50.425,179.886,6.374,149.192
C06165=1138.149,26.066,-50.439,179.888,6.375,149.191
C06166=1138.144,26.316,-50.454,179.891,6.377,149.191
C06167=1138.139,26.566,-50.468,179.894,6.377,149.190
C06168=1138.134,26.816,-50.482,179.896,6.378,149.190
C06169=1138.128,27.084,-50.498,179.899,6.379,149.189
C06170=1138.122,27.353,-50.513,179.902,6.381,149.189
C06171=1138.117,27.622,-50.528,179.905,6.381,149.188
C06172=1138.111,27.891,-50.545,179.907,6.383,149.188
C06173=1138.107,28.141,-50.559,179.910,6.383,149.187
C06174=1138.102,28.390,-50.573,179.912,6.384,149.186
C06175=1138.097,28.640,-50.587,179.915,6.386,149.186
C06176=1138.091,28.889,-50.602,179.918,6.386,149.185
C06177=1138.086,29.138,-50.616,179.920,6.388,149.185
C06178=1138.081,29.388,-50.631,179.923,6.388,149.184
C06179=1138.076,29.638,-50.645,179.926,6.390,149.184
C06180=1138.071,29.887,-50.660,179.928,6.391,149.183
C06181=1138.066,30.137,-50.675,179.931,6.391,149.183
C06182=1138.061,30.387,-50.689,179.933,6.393,149.182
C06183=1138.056,30.636,-50.703,179.936,6.393,149.182
C06184=1138.051,30.886,-50.719,179.939,6.395,149.181
C06185=1138.046,31.135,-50.733,179.941,6.396,149.181
C06186=1138.040,31.384,-50.747,179.943,6.396,149.180
C06187=1138.036,31.633,-50.762,179.946,6.398,149.179
C06188=1138.031,31.883,-50.776,179.949,6.398,149.179
C06189=1138.025,32.133,-50.791,179.951,6.400,149.178
C06190=1138.020,32.382,-50.806,179.954,6.400,149.178
C06191=1138.015,32.632,-50.821,179.957,6.402,149.177
C06192=1138.010,32.882,-50.835,179.959,6.403,149.177
C06193=1138.005,33.131,-50.850,179.962,6.403,149.176
C06194=1138.000,33.381,-50.865,179.964,6.405,149.176
C06195=1137.995,33.630,-50.880,179.967,6.406,149.175
C06196=1137.990,33.880,-50.895,179.970,6.407,149.175
C06197=1137.985,34.130,-50.909,179.972,6.408,149.174
C06198=1137.980,34.379,-50.924,179.975,6.410,149.174
C06199=1137.975,34.628,-50.938,179.977,6.410,149.173
C06200=1137.970,34.878,-50.954,179.980,6.412,149.173
C06201=1137.965,35.128,-50.968,179.983,6.412,149.172
C06202=1137.960,35.377,-50.983,179.985,6.413,149.171
C06203=1137.955,35.627,-50.998,179.988,6.415,149.171
C06204=1137.950,35.876,-51.013,179.990,6.415,149.170
C06205=1137.945,36.125,-51.027,179.993,6.417,149.170
C06206=1137.940,36.375,-51.043,179.995,6.417,149.169
C06207=1137.935,36.625,-51.057,179.999,6.419,149.169
C06208=1137.929,36.874,-51.073,-179.999,6.419,149.168
C06209=1137.924,37.124,-51.087,-179.997,6.421,149.168
C06210=1137.920,37.373,-51.102,-179.994,6.422,149.167
C06211=1137.914,37.623,-51.117,-179.991,6.423,149.167
C06212=1137.909,37.872,-51.132,-179.989,6.424,149.166
C06213=1137.904,38.122,-51.146,-179.986,6.425,149.166
C06214=1137.899,38.371,-51.162,-179.984,6.426,149.165
C06215=1137.894,38.620,-51.177,-179.981,6.427,149.165
C06216=1137.889,38.870,-51.191,-179.978,6.428,149.164
C06217=1137.884,39.119,-51.206,-179.976,6.429,149.164
C06218=1137.878,39.369,-51.221,-179.973,6.431,149.163
C06219=1137.874,39.618,-51.236,-179.971,6.431,149.162
C06220=1137.869,39.867,-51.251,-179.968,6.433,149.162
C06221=1137.863,40.117,-51.266,-179.966,6.434,149.162
C06222=1137.859,40.367,-51.281,-179.962,6.435,149.161
C06223=1137.853,40.616,-51.297,-179.960,6.436,149.160
C06224=1137.848,40.866,-51.311,-179.958,6.437,149.160
C06225=1137.843,41.115,-51.327,-179.955,6.438,149.159
C06226=1137.839,41.365,-51.342,-179.952,6.439,149.159
C06227=1137.833,41.615,-51.357,-179.950,6.440,149.158
C06228=1137.828,41.864,-51.372,-179.947,6.441,149.158
C06229=1137.823,42.113,-51.387,-179.945,6.442,149.157
C06230=1137.818,42.362,-51.402,-179.942,6.444,149.157
C06231=1137.813,42.612,-51.417,-179.939,6.444,149.156
C06232=1137.808,42.862,-51.432,-179.936,6.446,149.156
C06233=1137.803,43.111,-51.448,-179.934,6.447,149.155
C06234=1137.798,43.360,-51.463,-179.931,6.448,149.155
C06235=1137.793,43.611,-51.478,-179.929,6.449,149.154
C06236=1137.788,43.860,-51.493,-179.926,6.451,149.154
C06237=1137.783,44.109,-51.509,-179.923,6.451,149.153
C06238=1137.778,44.359,-51.524,-179.921,6.453,149.153
C06239=1137.773,44.608,-51.539,-179.918,6.453,149.152
C06240=1137.768,44.857,-51.555,-179.915,6.455,149.152
C06241=1137.763,45.107,-51.569,-179.913,6.456,149.151
C06242=1137.758,45.357,-51.585,-179.910,6.457,149.151
C06243=1137.753,45.606,-51.600,-179.908,6.458,149.150
C06244=1137.748,45.855,-51.616,-179.905,6.459,149.149
C06245=1137.742,46.105,-51.631,-179.903,6.460,149.149
C06246=1137.738,46.354,-51.646,-179.900,6.462,149.149
C06247=1137.733,46.604,-51.662,-179.897,6.463,149.148
C06248=1137.728,46.853,-51.677,-179.895,6.464,149.147
C06249=1137.723,47.103,-51.692,-179.892,6.465,149.147
C06250=1137.717,47.353,-51.708,-179.889,6.466,149.146
C06251=1137.713,47.602,-51.723,-179.886,6.468,149.146
C06252=1137.708,47.852,-51.739,-179.884,6.468,149.145
C06253=1137.702,48.101,-51.754,-179.881,6.470,149.145
C06254=1137.698,48.350,-51.769,-179.879,6.471,149.144
C06255=1137.692,48.600,-51.785,-179.876,6.472,149.144
C06256=1137.687,48.849,-51.800,-179.873,6.473,149.143
C06257=1137.683,49.099,-51.816,-179.871,6.474,149.143
C06258=1137.678,49.348,-51.831,-179.868,6.476,149.142
C06259=1137.672,49.598,-51.847,-179.865,6.476,149.142
C06260=1137.667,49.847,-51.862,-179.863,6.478,149.141
C06261=1137.663,50.097,-51.878,-179.860,6.479,149.141
C06262=1137.657,50.346,-51.893,-179.857,6.480,149.140
C06263=1137.652,50.596,-51.909,-179.855,6.481,149.140
C06264=1137.647,50.845,-51.924,-179.852,6.483,149.139
C06265=1137.642,51.095,-51.940,-179.850,6.483,149.139
C06266=1137.637,51.344,-51.956,-179.847,6.485,149.138
C06267=1137.632,51.593,-51.972,-179.844,6.486,149.138
C06268=1137.628,51.843,-51.987,-179.842,6.487,149.137
C06269=1137.623,52.092,-52.003,-179.839,6.488,149.137
C06270=1137.617,52.342,-52.018,-179.837,6.489,149.136
C06271=1137.612,52.591,-52.034,-179.834,6.491,149.136
C06272=1137.608,52.841,-52.049,-179.831,6.491,149.135
C06273=1137.602,53.109,-52.066,-179.828,6.493,149.135
C06274=1137.597,53.378,-52.083,-179.825,6.494,149.134
C06275=1137.591,53.646,-52.100,-179.822,6.496,149.133
C06276=1137.586,53.915,-52.117,-179.819,6.497,149.133
C06277=1137.581,54.165,-52.133,-179.817,6.498,149.132
C06278=1137.575,54.414,-52.149,-179.814,6.500,149.132
C06279=1137.570,54.664,-52.164,-179.812,6.500,149.131
C06280=1137.566,54.913,-52.181,-179.809,6.502,149.131
C06281=1137.561,55.162,-52.196,-179.807,6.503,149.130
C06282=1137.555,55.412,-52.212,-179.804,6.504,149.130
C06283=1137.551,55.662,-52.228,-179.801,6.505,149.129
C06284=1137.546,55.911,-52.244,-179.799,6.506,149.129
C06285=1137.540,56.160,-52.260,-179.796,6.508,149.128
C06286=1137.535,56.410,-52.276,-179.793,6.508,149.128
C06287=1137.530,56.659,-52.291,-179.790,6.510,149.127
C06288=1137.526,56.908,-52.307,-179.788,6.512,149.127
C06289=1137.521,57.158,-52.323,-179.785,6.513,149.126
C06290=1137.516,57.407,-52.338,-179.782,6.514,149.126
C06291=1137.511,57.657,-52.355,-179.780,6.515,149.125
C06292=1137.506,57.906,-52.371,-179.777,6.516,149.125
C06293=1137.500,58.156,-52.386,-179.774,6.518,149.124
C06294=1137.496,58.405,-52.403,-179.772,6.518,149.124
C06295=1137.490,58.655,-52.418,-179.769,6.520,149.123
C06296=1137.486,58.905,-52.434,-179.766,6.522,149.123
C06297=1137.481,59.153,-52.451,-179.764,6.522,149.122
C06298=1137.475,59.403,-52.466,-179.761,6.524,149.122
C06299=1137.471,59.652,-52.483,-179.759,6.525,149.121
C06300=1137.465,59.902,-52.499,-179.756,6.526,149.121
C06301=1137.461,60.151,-52.515,-179.753,6.528,149.120
C06302=1137.455,60.401,-52.531,-179.751,6.528,149.120
C06303=1137.451,60.651,-52.547,-179.748,6.530,149.119
C06304=1137.446,60.900,-52.563,-179.745,6.531,149.119
C06305=1137.440,61.149,-52.579,-179.743,6.532,149.118
C06306=1137.436,61.398,-52.595,-179.740,6.534,149.118
C06307=1137.430,61.648,-52.611,-179.737,6.535,149.117
C06308=1137.426,61.897,-52.628,-179.734,6.536,149.117
C06309=1137.420,62.147,-52.643,-179.732,6.538,149.116
C06310=1137.416,62.396,-52.660,-179.730,6.538,149.116
C06311=1137.411,62.646,-52.675,-179.726,6.540,149.115
C06312=1137.406,62.895,-52.692,-179.724,6.541,149.115
C06313=1137.401,63.144,-52.708,-179.721,6.542,149.114
C06314=1137.396,63.394,-52.724,-179.718,6.543,149.114
C06315=1137.391,63.643,-52.741,-179.715,6.545,149.113
C06316=1137.386,63.893,-52.757,-179.713,6.546,149.113
C06317=1137.381,64.142,-52.774,-179.711,6.548,149.112
C06318=1137.376,64.392,-52.789,-179.707,6.549,149.112
C06319=1137.371,64.641,-52.806,-179.705,6.550,149.111
C06320=1137.366,64.890,-52.822,-179.702,6.551,149.111
C06321=1137.361,65.140,-52.838,-179.700,6.553,149.110
C06322=1137.356,65.389,-52.855,-179.697,6.553,149.110
C06323=1137.351,65.638,-52.871,-179.694,6.555,149.109
C06324=1137.346,65.888,-52.887,-179.691,6.557,149.109
C06325=1137.341,66.137,-52.904,-179.689,6.557,149.108
C06326=1137.336,66.387,-52.921,-179.686,6.559,149.108
C06327=1137.331,66.637,-52.936,-179.683,6.561,149.107
C06328=1137.326,66.886,-52.953,-179.681,6.561,149.107
C06329=1137.322,67.135,-52.969,-179.678,6.563,149.106
C06330=1137.316,67.384,-52.985,-179.675,6.564,149.106
C06331=1137.311,67.634,-53.002,-179.673,6.565,149.105
C06332=1137.306,67.883,-53.019,-179.670,6.567,149.105
C06333=1137.302,68.133,-53.035,-179.667,6.568,149.104
C06334=1137.297,68.383,-53.051,-179.665,6.569,149.104
C06335=1137.292,68.631,-53.068,-179.662,6.571,149.103
C06336=1137.287,68.881,-53.085,-179.659,6.572,149.103
C06337=1137.281,69.130,-53.101,-179.656,6.573,149.102
C06338=1137.277,69.379,-53.118,-179.654,6.574,149.102
C06339=1137.272,69.630,-53.134,-179.651,6.576,149.101
C06340=1137.266,69.879,-53.151,-179.649,6.578,149.101
C06341=1137.262,70.128,-53.167,-179.646,6.578,149.100
C06342=1137.257,70.377,-53.184,-179.643,6.580,149.100
C06343=1137.252,70.627,-53.201,-179.640,6.581,149.099
C06344=1137.247,70.876,-53.218,-179.638,6.582,149.099
C06345=1137.242,71.126,-53.233,-179.635,6.584,149.098
C06346=1137.237,71.375,-53.250,-179.632,6.585,149.098
C06347=1137.232,71.625,-53.267,-179.630,6.587,149.097
C06348=1137.227,71.874,-53.283,-179.627,6.588,149.097
C06349=1137.222,72.123,-53.300,-179.624,6.589,149.096
C06350=1137.217,72.373,-53.317,-179.621,6.591,149.096
C06351=1137.212,72.622,-53.334,-179.619,6.592,149.096
C06352=1137.208,72.871,-53.350,-179.616,6.593,149.095
C06353=1137.202,73.121,-53.368,-179.613,6.594,149.094
C06354=1137.197,73.370,-53.384,-179.611,6.596,149.094
C06355=1137.192,73.620,-53.401,-179.608,6.597,149.094
C06356=1137.188,73.869,-53.418,-179.606,6.599,149.093
C06357=1137.183,74.118,-53.434,-179.602,6.600,149.092
C06358=1137.177,74.368,-53.451,-179.600,6.602,149.092
C06359=1137.173,74.617,-53.468,-179.597,6.602,149.092
C06360=1137.168,74.866,-53.484,-179.595,6.604,149.091
C06361=1137.163,75.116,-53.502,-179.592,6.605,149.091
C06362=1137.158,75.365,-53.518,-179.589,6.607,149.090
C06363=1137.152,75.614,-53.535,-179.587,6.608,149.090
C06364=1137.148,75.864,-53.552,-179.584,6.609,149.089
C06365=1137.143,76.114,-53.569,-179.581,6.611,149.089
C06366=1137.138,76.363,-53.586,-179.578,6.612,149.088
C06367=1137.133,76.612,-53.602,-179.576,6.613,149.088
C06368=1137.128,76.862,-53.619,-179.573,6.615,149.087
C06369=1137.124,77.110,-53.637,-179.570,6.617,149.087
C06370=1137.118,77.360,-53.654,-179.567,6.618,149.086
C06371=1137.113,77.609,-53.670,-179.565,6.619,149.086
C06372=1137.108,77.859,-53.688,-179.562,6.620,149.085
C06373=1137.104,78.108,-53.704,-179.559,6.622,149.085
C06374=1137.098,78.358,-53.721,-179.556,6.623,149.084
C06375=1137.094,78.606,-53.738,-179.554,6.624,149.084
C06376=1137.088,78.856,-53.756,-179.551,6.626,149.083
C06377=1137.083,79.125,-53.774,-179.549,6.627,149.083
C06378=1137.078,79.393,-53.792,-179.545,6.629,149.082
C06379=1137.072,79.662,-53.811,-179.543,6.630,149.082
C06380=1137.068,79.930,-53.829,-179.539,6.632,149.081
C06381=1137.062,80.179,-53.846,-179.537,6.633,149.081
C06382=1137.058,80.428,-53.863,-179.534,6.635,149.080
C06383=1137.053,80.678,-53.880,-179.532,6.636,149.080
C06384=1137.047,80.928,-53.898,-179.529,6.638,149.080
C06385=1137.043,81.177,-53.914,-179.526,6.639,149.079
C06386=1137.038,81.426,-53.932,-179.523,6.640,149.078
C06387=1137.033,81.675,-53.949,-179.520,6.642,149.078
C06388=1137.028,81.925,-53.966,-179.518,6.643,149.078
C06389=1137.023,82.174,-53.984,-179.515,6.645,149.077
C06390=1137.018,82.424,-54.001,-179.512,6.646,149.077
C06391=1137.013,82.674,-54.018,-179.509,6.648,149.076
C06392=1137.008,82.923,-54.036,-179.507,6.649,149.076
C06393=1137.003,83.171,-54.052,-179.504,6.650,149.075
C06394=1136.998,83.421,-54.069,-179.502,6.652,149.075
C06395=1136.994,83.670,-54.087,-179.498,6.653,149.074
C06396=1136.988,83.920,-54.104,-179.496,6.655,149.074
C06397=1136.984,84.169,-54.122,-179.493,6.656,149.073
C06398=1136.979,84.419,-54.139,-179.491,6.657,149.073
C06399=1136.974,84.668,-54.157,-179.488,6.659,149.072
C06400=1136.969,84.918,-54.174,-179.485,6.660,149.072
C06401=1136.964,85.167,-54.191,-179.482,6.662,149.071
C06402=1136.959,85.416,-54.208,-179.479,6.664,149.071
C06403=1136.954,85.665,-54.226,-179.477,6.664,149.071
C06404=1136.949,85.914,-54.244,-179.475,6.666,149.070
C06405=1136.944,86.164,-54.260,-179.471,6.667,149.069
C06406=1136.939,86.413,-54.278,-179.469,6.669,149.069
C06407=1136.934,86.663,-54.295,-179.466,6.671,149.069
C06408=1136.929,86.912,-54.313,-179.463,6.672,149.068
C06409=1136.925,87.161,-54.331,-179.461,6.673,149.068
C06410=1136.920,87.411,-54.348,-179.458,6.674,149.067
C06411=1136.915,87.660,-54.366,-179.455,6.676,149.067
C06412=1136.910,87.910,-54.383,-179.452,6.678,149.066
C06413=1136.905,88.159,-54.401,-179.449,6.679,149.066
C06414=1136.900,88.408,-54.418,-179.447,6.681,149.065
C06415=1136.895,88.658,-54.436,-179.445,6.682,149.065
C06416=1136.891,88.907,-54.454,-179.441,6.683,149.064
C06417=1136.885,89.157,-54.471,-179.439,6.685,149.064
C06418=1136.880,89.406,-54.489,-179.436,6.687,149.064
C06419=1136.876,89.654,-54.506,-179.433,6.688,149.063
C06420=1136.870,89.904,-54.523,-179.430,6.690,149.063
C06421=1136.866,90.153,-54.541,-179.428,6.692,149.062
C06422=1136.861,90.402,-54.559,-179.425,6.692,149.062
C06423=1136.855,90.652,-54.577,-179.422,6.694,149.061
C06424=1136.850,90.901,-54.595,-179.420,6.695,149.061
C06425=1136.846,91.151,-54.613,-179.417,6.697,149.060
C06426=1136.842,91.400,-54.630,-179.414,6.699,149.060
C06427=1136.837,91.650,-54.648,-179.411,6.700,149.059
C06428=1136.832,91.899,-54.666,-179.408,6.702,149.059
C06429=1136.827,92.148,-54.684,-179.406,6.703,149.058
C06430=1136.822,92.398,-54.701,-179.403,6.704,149.058
C06431=1136.817,92.647,-54.719,-179.400,6.706,149.058
C06432=1136.812,92.896,-54.737,-179.398,6.708,149.057
C06433=1136.807,93.145,-54.755,-179.395,6.709,149.057
C06434=1136.802,93.394,-54.773,-179.392,6.711,149.056
C06435=1136.797,93.644,-54.790,-179.389,6.712,149.056
C06436=1136.792,93.893,-54.808,-179.386,6.714,149.055
C06437=1136.787,94.143,-54.826,-179.384,6.716,149.055
C06438=1136.782,94.392,-54.844,-179.381,6.716,149.054
C06439=1136.777,94.641,-54.862,-179.379,6.718,149.054
C06440=1136.772,94.890,-54.880,-179.375,6.719,149.053
C06441=1136.767,95.140,-54.897,-179.373,6.721,149.053
C06442=1136.762,95.389,-54.915,-179.370,6.723,149.053
C06443=1136.758,95.639,-54.934,-179.367,6.724,149.052
C06444=1136.753,95.888,-54.951,-179.364,6.726,149.052
C06445=1136.748,96.137,-54.969,-179.362,6.728,149.051
C06446=1136.743,96.386,-54.987,-179.359,6.729,149.051
C06447=1136.738,96.636,-55.005,-179.356,6.730,149.050
C06448=1136.733,96.885,-55.023,-179.354,6.732,149.050
C06449=1136.728,97.134,-55.041,-179.351,6.733,149.049
C06450=1136.723,97.383,-55.059,-179.348,6.735,149.049
C06451=1136.719,97.633,-55.078,-179.345,6.737,149.049
C06452=1136.714,97.882,-55.096,-179.343,6.738,149.048
C06453=1136.709,98.131,-55.114,-179.340,6.740,149.048
C06454=1136.704,98.381,-55.132,-179.337,6.741,149.047
C06455=1136.700,98.630,-55.150,-179.334,6.743,149.047
C06456=1136.695,98.879,-55.168,-179.331,6.745,149.046
C06457=1136.690,99.128,-55.186,-179.329,6.746,149.046
C06458=1136.685,99.378,-55.205,-179.326,6.748,149.045
C06459=1136.680,99.627,-55.223,-179.324,6.749,149.045
C06460=1136.675,99.877,-55.241,-179.321,6.750,149.045
C06461=1136.670,100.126,-55.258,-179.318,6.752,149.044
C06462=1136.665,100.374,-55.277,-179.315,6.753,149.043
C06463=1136.661,100.624,-55.296,-179.312,6.755,149.043
C06464=1136.656,100.873,-55.314,-179.310,6.757,149.043
C06465=1136.650,101.123,-55.332,-179.307,6.758,149.042
C06466=1136.646,101.372,-55.350,-179.304,6.760,149.042
C06467=1136.641,101.621,-55.368,-179.301,6.762,149.041
C06468=1136.636,101.871,-55.386,-179.299,6.763,149.041
C06469=1136.632,102.120,-55.405,-179.296,6.765,149.041
C06470=1136.626,102.369,-55.424,-179.293,6.766,149.040
C06471=1136.621,102.618,-55.442,-179.290,6.768,149.040
C06472=1136.617,102.868,-55.460,-179.287,6.770,149.039
C06473=1136.612,103.117,-55.478,-179.284,6.771,149.039
C06474=1136.607,103.366,-55.497,-179.282,6.773,149.038
C06475=1136.602,103.615,-55.515,-179.279,6.775,149.038
C06476=1136.597,103.865,-55.534,-179.276,6.776,149.037
C06477=1136.592,104.114,-55.552,-179.274,6.777,149.037
C06478=1136.588,104.363,-55.570,-179.271,6.779,149.037
C06479=1136.582,104.613,-55.589,-179.268,6.780,149.036
C06480=1136.578,104.862,-55.607,-179.265,6.782,149.036
C06481=1136.572,105.130,-55.628,-179.262,6.784,149.035
C06482=1136.567,105.399,-55.647,-179.259,6.786,149.035
C06483=1136.562,105.667,-55.667,-179.257,6.788,149.034
C06484=1136.556,105.935,-55.687,-179.253,6.789,149.034
C06485=1136.552,106.185,-55.706,-179.251,6.791,149.033
C06486=1136.547,106.434,-55.724,-179.248,6.792,149.033
C06487=1136.542,106.683,-55.742,-179.245,6.794,149.032
C06488=1136.538,106.933,-55.761,-179.242,6.796,149.032
C06489=1136.532,107.182,-55.780,-179.240,6.797,149.032
C06490=1136.528,107.431,-55.799,-179.237,6.799,149.031
C06491=1136.523,107.681,-55.817,-179.234,6.801,149.031
C06492=1136.518,107.929,-55.836,-179.231,6.803,149.030
C06493=1136.513,108.179,-55.854,-179.229,6.804,149.030
C06494=1136.509,108.428,-55.873,-179.226,6.806,149.029
C06495=1136.503,108.677,-55.892,-179.223,6.807,149.029
C06496=1136.498,108.926,-55.910,-179.220,6.809,149.029
C06497=1136.494,109.176,-55.930,-179.217,6.811,149.028
C06498=1136.489,109.425,-55.948,-179.215,6.812,149.028
C06499=1136.485,109.674,-55.967,-179.212,6.814,149.027
C06500=1136.479,109.924,-55.985,-179.209,6.816,149.027
C06501=1136.474,110.173,-56.004,-179.206,6.817,149.027
C06502=1136.470,110.422,-56.024,-179.204,6.819,149.026
C06503=1136.465,110.671,-56.041,-179.201,6.821,149.026
C06504=1136.459,110.920,-56.061,-179.198,6.822,149.025
C06505=1136.455,111.170,-56.079,-179.195,6.824,149.025
C06506=1136.450,111.419,-56.098,-179.193,6.826,149.024
C06507=1136.446,111.668,-56.117,-179.190,6.827,149.024
C06508=1136.440,111.918,-56.136,-179.187,6.829,149.023
C06509=1136.436,112.167,-56.155,-179.184,6.830,149.023
C06510=1136.431,112.416,-56.174,-179.181,6.832,149.023
C06511=1136.426,112.665,-56.192,-179.179,6.834,149.022
C06512=1136.421,112.914,-56.212,-179.176,6.835,149.022
C06513=1136.416,113.164,-56.230,-179.173,6.837,149.021
C06514=1136.412,113.413,-56.250,-179.170,6.839,149.021
C06515=1136.407,113.662,-56.268,-179.168,6.840,149.021
C06516=1136.402,113.912,-56.287,-179.165,6.842,149.020
C06517=1136.397,114.161,-56.307,-179.162,6.845,149.020
C06518=1136.392,114.409,-56.325,-179.159,6.846,149.019
C06519=1136.387,114.659,-56.345,-179.156,6.848,149.019
C06520=1136.382,114.908,-56.363,-179.153,6.850,149.019
C06521=1136.378,115.158,-56.383,-179.151,6.851,149.018
C06522=1136.372,115.407,-56.402,-179.148,6.853,149.018
C06523=1136.368,115.656,-56.421,-179.145,6.855,149.017
C06524=1136.363,115.905,-56.440,-179.143,6.856,149.017
C06525=1136.358,116.155,-56.459,-179.140,6.858,149.017
C06526=1136.353,116.403,-56.478,-179.137,6.860,149.016
C06527=1136.348,116.653,-56.498,-179.134,6.861,149.016
C06528=1136.344,116.902,-56.516,-179.131,6.863,149.015
C06529=1136.339,117.151,-56.536,-179.128,6.864,149.015
C06530=1136.334,117.400,-56.555,-179.126,6.866,149.014
C06531=1136.329,117.650,-56.574,-179.123,6.868,149.014
C06532=1136.325,117.899,-56.593,-179.120,6.869,149.013
C06533=1136.319,118.148,-56.612,-179.117,6.871,149.013
C06534=1136.315,118.398,-56.632,-179.114,6.874,149.013
C06535=1136.310,118.646,-56.651,-179.111,6.875,149.012
C06536=1136.305,118.896,-56.670,-179.109,6.877,149.012
C06537=1136.300,119.145,-56.690,-179.106,6.879,149.011
C06538=1136.296,119.394,-56.709,-179.103,6.880,149.011
C06539=1136.291,119.643,-56.728,-179.101,6.882,149.011
C06540=1136.286,119.893,-56.748,-179.098,6.884,149.010
C06541=1136.282,120.142,-56.767,-179.095,6.885,149.010
C06542=1136.276,120.391,-56.786,-179.092,6.887,149.009
C06543=1136.272,120.640,-56.806,-179.090,6.889,149.009
C06544=1136.266,120.889,-56.825,-179.087,6.890,149.009
C06545=1136.262,121.139,-56.845,-179.084,6.892,149.008
C06546=1136.258,121.388,-56.864,-179.081,6.895,149.008
C06547=1136.252,121.637,-56.883,-179.078,6.896,149.007
C06548=1136.248,121.886,-56.903,-179.075,6.898,149.007
C06549=1136.242,122.135,-56.922,-179.073,6.900,149.007
C06550=1136.237,122.385,-56.942,-179.070,6.901,149.006
C06551=1136.233,122.634,-56.961,-179.067,6.903,149.006
C06552=1136.228,122.883,-56.980,-179.064,6.905,149.005
C06553=1136.224,123.132,-57.000,-179.062,6.906,149.005
C06554=1136.219,123.381,-57.020,-179.059,6.908,149.005
C06555=1136.214,123.630,-57.039,-179.056,6.911,149.004
C06556=1136.209,123.880,-57.059,-179.053,6.912,149.004
C06557=1136.205,124.129,-57.078,-179.050,6.914,149.003
C06558=1136.199,124.378,-57.097,-179.047,6.916,149.003
C06559=1136.195,124.627,-57.118,-179.045,6.917,149.003
C06560=1136.190,124.877,-57.137,-179.042,6.919,149.002
C06561=1136.185,125.125,-57.157,-179.039,6.921,149.002
C06562=1136.180,125.375,-57.176,-179.037,6.922,149.001
C06563=1136.175,125.625,-57.196,-179.033,6.925,149.001
C06564=1136.170,125.873,-57.216,-179.031,6.927,149.001
C06565=1136.166,126.122,-57.236,-179.028,6.928,149.000
C06566=1136.161,126.372,-57.255,-179.025,6.930,149.000
C06567=1136.156,126.622,-57.275,-179.022,6.932,148.999
C06568=1136.152,126.869,-57.294,-179.020,6.933,148.999
C06569=1136.147,127.119,-57.314,-179.017,6.935,148.999
C06570=1136.142,127.369,-57.334,-179.014,6.938,148.998
C06571=1136.137,127.617,-57.354,-179.011,6.939,148.998
C06572=1136.133,127.866,-57.373,-179.008,6.941,148.997
C06573=1136.128,128.116,-57.393,-179.005,6.943,148.997
C06574=1136.123,128.365,-57.413,-179.003,6.945,148.997
C06575=1136.118,128.614,-57.433,-179.000,6.946,148.996
C06576=1136.114,128.863,-57.453,-178.998,6.948,148.996
C06577=1136.109,129.112,-57.473,-178.994,6.951,148.996
C06578=1136.104,129.362,-57.492,-178.992,6.952,148.995
C06579=1136.098,129.610,-57.513,-178.989,6.954,148.995
C06580=1136.094,129.860,-57.533,-178.986,6.956,148.994
C06581=1136.089,130.109,-57.553,-178.984,6.957,148.994
C06582=1136.084,130.359,-57.573,-178.981,6.959,148.994
C06583=1136.080,130.607,-57.593,-178.977,6.961,148.993
C06584=1136.075,130.856,-57.612,-178.975,6.963,148.993
C06585=1136.070,131.125,-57.633,-178.972,6.965,148.993
C06586=1136.064,131.393,-57.656,-178.969,6.967,148.992
C06587=1136.060,131.662,-57.677,-178.966,6.969,148.992
C06588=1136.054,131.931,-57.699,-178.963,6.971,148.991
C06589=1136.049,132.180,-57.719,-178.960,6.973,148.991
C06590=1136.045,132.429,-57.739,-178.957,6.975,148.991
C06591=1136.040,132.678,-57.759,-178.955,6.977,148.990
C06592=1136.036,132.927,-57.779,-178.952,6.978,148.990
C06593=1136.030,133.176,-57.799,-178.949,6.980,148.989
C06594=1136.025,133.425,-57.820,-178.946,6.983,148.989
C06595=1136.021,133.675,-57.839,-178.943,6.984,148.989
C06596=1136.016,133.924,-57.860,-178.940,6.986,148.988
C06597=1136.012,134.173,-57.880,-178.938,6.988,148.988
C06598=1136.007,134.423,-57.900,-178.935,6.989,148.987
C06599=1136.003,134.671,-57.920,-178.932,6.992,148.987
C06600=1135.997,134.920,-57.941,-178.929,6.994,148.987
C06601=1135.992,135.170,-57.960,-178.927,6.996,148.986
C06602=1135.988,135.419,-57.981,-178.924,6.997,148.986
C06603=1135.983,135.667,-58.001,-178.921,6.999,148.986
C06604=1135.978,135.917,-58.021,-178.918,7.001,148.985
C06605=1135.973,136.166,-58.042,-178.915,7.003,148.985
C06606=1135.969,136.415,-58.062,-178.912,7.005,148.985
C06607=1135.964,136.664,-58.082,-178.910,7.007,148.984
C06608=1135.959,136.914,-58.103,-178.906,7.009,148.984
C06609=1135.954,137.163,-58.123,-178.904,7.011,148.983
C06610=1135.950,137.412,-58.143,-178.901,7.012,148.983
C06611=1135.944,137.661,-58.164,-178.898,7.014,148.983
C06612=1135.939,137.910,-58.184,-178.896,7.016,148.982
C06613=1135.935,138.159,-58.204,-178.893,7.019,148.982
C06614=1135.931,138.408,-58.224,-178.890,7.020,148.982
C06615=1135.925,138.657,-58.245,-178.887,7.022,148.981
C06616=1135.921,138.906,-58.266,-178.884,7.024,148.981
C06617=1135.917,139.155,-58.286,-178.881,7.026,148.980
C06618=1135.911,139.404,-58.307,-178.878,7.028,148.980
C06619=1135.907,139.654,-58.327,-178.876,7.030,148.980
C06620=1135.902,139.903,-58.347,-178.873,7.031,148.979
C06621=1135.897,140.152,-58.368,-178.870,7.034,148.979
C06622=1135.893,140.401,-58.388,-178.867,7.036,148.979
C06623=1135.887,140.650,-58.409,-178.865,7.038,148.978
C06624=1135.883,140.899,-58.430,-178.862,7.039,148.978
C06625=1135.879,141.148,-58.450,-178.859,7.042,148.978
C06626=1135.873,141.398,-58.471,-178.856,7.044,148.977
C06627=1135.869,141.647,-58.491,-178.853,7.045,148.977
C06628=1135.864,141.896,-58.512,-178.851,7.047,148.976
C06629=1135.859,142.145,-58.533,-178.847,7.049,148.976
C06630=1135.854,142.394,-58.554,-178.845,7.051,148.976
C06631=1135.850,142.643,-58.574,-178.842,7.053,148.975
C06632=1135.845,142.892,-58.595,-178.840,7.055,148.975
C06633=1135.840,143.141,-58.615,-178.836,7.057,148.975
C06634=1135.836,143.391,-58.636,-178.833,7.059,148.974
C06635=1135.831,143.640,-58.657,-178.831,7.061,148.974
C06636=1135.827,143.889,-58.678,-178.827,7.063,148.974
C06637=1135.822,144.138,-58.699,-178.825,7.065,148.973
C06638=1135.817,144.387,-58.720,-178.823,7.067,148.973
C06639=1135.812,144.636,-58.741,-178.820,7.069,148.973
C06640=1135.808,144.885,-58.761,-178.816,7.071,148.972
C06641=1135.803,145.134,-58.782,-178.814,7.073,148.972
C06642=1135.798,145.383,-58.802,-178.811,7.075,148.971
C06643=1135.793,145.632,-58.823,-178.808,7.078,148.971
C06644=1135.788,145.881,-58.845,-178.805,7.079,148.971
C06645=1135.784,146.130,-58.865,-178.803,7.081,148.971
C06646=1135.779,146.380,-58.887,-178.800,7.083,148.970
C06647=1135.775,146.629,-58.907,-178.797,7.085,148.970
C06648=1135.769,146.878,-58.928,-178.794,7.087,148.969
C06649=1135.765,147.127,-58.950,-178.791,7.089,148.969
C06650=1135.760,147.376,-58.970,-178.788,7.091,148.969
C06651=1135.755,147.625,-58.991,-178.786,7.093,148.968
C06652=1135.750,147.874,-59.011,-178.783,7.095,148.968
C06653=1135.746,148.123,-59.033,-178.780,7.097,148.968
C06654=1135.741,148.372,-59.054,-178.777,7.099,148.967
C06655=1135.737,148.621,-59.075,-178.775,7.101,148.967
C06656=1135.732,148.870,-59.096,-178.772,7.103,148.967
C06657=1135.727,149.119,-59.117,-178.769,7.105,148.966
C06658=1135.722,149.368,-59.138,-178.766,7.107,148.966
C06659=1135.718,149.618,-59.160,-178.763,7.109,148.966
C06660=1135.713,149.867,-59.181,-178.760,7.111,148.965
C06661=1135.708,150.116,-59.201,-178.758,7.113,148.965
C06662=1135.703,150.364,-59.223,-178.755,7.115,148.965
C06663=1135.698,150.614,-59.244,-178.752,7.118,148.964
C06664=1135.694,150.863,-59.266,-178.749,7.119,148.964
C06665=1135.690,151.112,-59.286,-178.746,7.121,148.964
C06666=1135.685,151.361,-59.308,-178.743,7.124,148.963
C06667=1135.679,151.610,-59.329,-178.741,7.126,148.963
C06668=1135.675,151.859,-59.349,-178.738,7.127,148.963
C06669=1135.671,152.108,-59.371,-178.735,7.130,148.962
C06670=1135.666,152.357,-59.392,-178.732,7.131,148.962
C06671=1135.661,152.606,-59.414,-178.729,7.134,148.962
C06672=1135.656,152.855,-59.435,-178.726,7.136,148.961
C06673=1135.652,153.104,-59.456,-178.724,7.138,148.961
C06674=1135.647,153.353,-59.478,-178.720,7.140,148.961
C06675=1135.642,153.602,-59.499,-178.718,7.142,148.960
C06676=1135.637,153.851,-59.521,-178.716,7.144,148.960
C06677=1135.633,154.101,-59.542,-178.712,7.147,148.960
C06678=1135.628,154.349,-59.563,-178.710,7.148,148.959
C06679=1135.623,154.598,-59.584,-178.707,7.150,148.959
C06680=1135.618,154.847,-59.606,-178.704,7.153,148.959
C06681=1135.614,155.096,-59.628,-178.701,7.155,148.958
C06682=1135.609,155.346,-59.649,-178.699,7.156,148.958
C06683=1135.604,155.594,-59.670,-178.695,7.159,148.958
C06684=1135.600,155.844,-59.693,-178.693,7.161,148.958
C06685=1135.595,156.093,-59.713,-178.690,7.163,148.957
C06686=1135.590,156.341,-59.735,-178.687,7.165,148.957
C06687=1135.586,156.591,-59.757,-178.684,7.167,148.956
C06688=1135.581,156.840,-59.778,-178.681,7.169,148.956
C06689=1135.576,157.109,-59.802,-178.679,7.171,148.956
C06690=1135.571,157.378,-59.824,-178.675,7.174,148.956
C06691=1135.566,157.647,-59.848,-178.672,7.176,148.955
C06692=1135.561,157.915,-59.871,-178.669,7.178,148.955
C06693=1135.556,158.164,-59.893,-178.666,7.181,148.954
C06694=1135.552,158.414,-59.914,-178.663,7.182,148.954
C06695=1135.547,158.663,-59.936,-178.661,7.185,148.954
C06696=1135.542,158.911,-59.958,-178.658,7.187,148.954
C06697=1135.538,159.161,-59.980,-178.655,7.189,148.953
C06698=1135.533,159.409,-60.001,-178.652,7.191,148.953
C06699=1135.528,159.659,-60.022,-178.650,7.193,148.953
C06700=1135.523,159.908,-60.044,-178.646,7.196,148.952
C06701=1135.519,160.157,-60.066,-178.644,7.197,148.952
C06702=1135.514,160.406,-60.088,-178.641,7.199,148.952
C06703=1135.509,160.654,-60.110,-178.638,7.202,148.951
C06704=1135.505,160.904,-60.132,-178.635,7.204,148.951
C06705=1135.500,161.152,-60.154,-178.632,7.206,148.951
C06706=1135.495,161.401,-60.176,-178.630,7.208,148.950
C06707=1135.490,161.651,-60.198,-178.627,7.210,148.950
C06708=1135.486,161.899,-60.220,-178.624,7.212,148.950
C06709=1135.481,162.149,-60.242,-178.621,7.214,148.949
C06710=1135.476,162.397,-60.263,-178.618,7.217,148.949
C06711=1135.472,162.647,-60.285,-178.616,7.219,148.949
C06712=1135.467,162.895,-60.307,-178.612,7.221,148.948
C06713=1135.463,163.145,-60.329,-178.610,7.223,148.948
C06714=1135.458,163.393,-60.351,-178.607,7.225,148.948
C06715=1135.454,163.643,-60.373,-178.604,7.228,148.948
C06716=1135.448,163.892,-60.395,-178.601,7.229,148.947
C06717=1135.444,164.141,-60.417,-178.598,7.232,148.947
C06718=1135.439,164.390,-60.439,-178.596,7.234,148.947
C06719=1135.435,164.639,-60.461,-178.592,7.236,148.946
C06720=1135.430,164.888,-60.483,-178.590,7.238,148.946
C06721=1135.426,165.137,-60.505,-178.587,7.241,148.946
C06722=1135.420,165.386,-60.527,-178.584,7.243,148.945
C06723=1135.416,165.635,-60.549,-178.582,7.245,148.945
C06724=1135.411,165.883,-60.571,-178.579,7.247,148.945
C06725=1135.407,166.133,-60.593,-178.576,7.249,148.945
C06726=1135.402,166.381,-60.615,-178.573,7.252,148.944
C06727=1135.397,166.631,-60.638,-178.570,7.254,148.944
C06728=1135.392,166.880,-60.659,-178.567,7.256,148.944
C06729=1135.388,167.128,-60.682,-178.565,7.258,148.944
C06730=1135.383,167.377,-60.704,-178.562,7.261,148.943
C06731=1135.378,167.627,-60.726,-178.559,7.262,148.943
C06732=1135.374,167.875,-60.748,-178.556,7.265,148.943
C06733=1135.370,168.124,-60.771,-178.553,7.267,148.942
C06734=1135.365,168.374,-60.794,-178.550,7.270,148.942
C06735=1135.360,168.622,-60.815,-178.548,7.272,148.942
C06736=1135.355,168.872,-60.837,-178.544,7.274,148.941
C06737=1135.350,169.120,-60.860,-178.542,7.276,148.941
C06738=1135.346,169.369,-60.882,-178.539,7.279,148.941
C06739=1135.342,169.619,-60.904,-178.536,7.280,148.941
C06740=1135.336,169.867,-60.927,-178.533,7.283,148.940
C06741=1135.332,170.116,-60.949,-178.531,7.285,148.940
C06742=1135.327,170.365,-60.971,-178.528,7.287,148.940
C06743=1135.322,170.614,-60.994,-178.525,7.289,148.939
C06744=1135.318,170.863,-61.016,-178.522,7.291,148.939
C06745=1135.314,171.111,-61.039,-178.519,7.294,148.939
C06746=1135.309,171.361,-61.062,-178.516,7.296,148.938
C06747=1135.304,171.610,-61.083,-178.514,7.299,148.938
C06748=1135.299,171.859,-61.107,-178.511,7.300,148.938
C06749=1135.295,172.108,-61.129,-178.508,7.303,148.938
C06750=1135.290,172.356,-61.151,-178.505,7.306,148.937
C06751=1135.285,172.606,-61.174,-178.502,7.307,148.937
C06752=1135.281,172.854,-61.196,-178.499,7.310,148.937
C06753=1135.276,173.103,-61.219,-178.497,7.312,148.937
C06754=1135.272,173.352,-61.241,-178.493,7.314,148.936
C06755=1135.267,173.602,-61.264,-178.491,7.317,148.936
C06756=1135.263,173.850,-61.287,-178.488,7.319,148.936
C06757=1135.257,174.099,-61.310,-178.486,7.321,148.936
C06758=1135.253,174.348,-61.332,-178.482,7.324,148.935
C06759=1135.248,174.597,-61.355,-178.480,7.325,148.935
C06760=1135.244,174.846,-61.377,-178.477,7.328,148.935
C06761=1135.239,175.095,-61.400,-178.474,7.330,148.934
C06762=1135.235,175.343,-61.423,-178.471,7.333,148.934
C06763=1135.230,175.593,-61.446,-178.468,7.335,148.934
C06764=1135.225,175.841,-61.468,-178.465,7.337,148.934
C06765=1135.220,176.091,-61.491,-178.463,7.339,148.933
C06766=1135.216,176.340,-61.514,-178.460,7.342,148.933
C06767=1135.211,176.588,-61.537,-178.457,7.344,148.933
C06768=1135.206,176.837,-61.560,-178.454,7.346,148.933
C06769=1135.202,177.086,-61.582,-178.451,7.349,148.932
C06770=1135.197,177.335,-61.605,-178.449,7.351,148.932
C06771=1135.193,177.584,-61.628,-178.445,7.353,148.932
C06772=1135.188,177.833,-61.650,-178.443,7.356,148.932
C06773=1135.184,178.082,-61.673,-178.440,7.358,148.931
C06774=1135.179,178.331,-61.696,-178.437,7.360,148.931
C06775=1135.174,178.580,-61.720,-178.434,7.363,148.931
C06776=1135.171,178.828,-61.743,-178.432,7.364,148.930
C06777=1135.165,179.077,-61.765,-178.429,7.367,148.930
C06778=1135.160,179.326,-61.788,-178.425,7.370,148.930
C06779=1135.156,179.575,-61.811,-178.423,7.372,148.930
C06780=1135.152,179.824,-61.834,-178.420,7.374,148.929
C06781=1135.147,180.073,-61.858,-178.418,7.376,148.929
C06782=1135.142,180.321,-61.880,-178.414,7.379,148.929
C06783=1135.138,180.570,-61.903,-178.412,7.381,148.929
C06784=1135.133,180.820,-61.926,-178.409,7.384,148.928
C06785=1135.129,181.069,-61.949,-178.406,7.386,148.928
C06786=1135.124,181.318,-61.972,-178.403,7.388,148.928
C06787=1135.119,181.567,-61.996,-178.400,7.391,148.928
C06788=1135.115,181.816,-62.019,-178.398,7.393,148.927
C06789=1135.110,182.064,-62.041,-178.395,7.395,148.927
C06790=1135.105,182.313,-62.065,-178.392,7.398,148.927
C06791=1135.101,182.562,-62.088,-178.389,7.400,148.927
C06792=1135.096,182.811,-62.111,-178.386,7.403,148.926
C06793=1135.091,183.080,-62.136,-178.383,7.405,148.926
C06794=1135.086,183.349,-62.162,-178.380,7.408,148.926
C06795=1135.082,183.620,-62.187,-178.377,7.410,148.926
C06796=1135.076,183.890,-62.212,-178.374,7.413,148.925
C06797=1135.072,184.139,-62.235,-178.371,7.415,148.925
C06798=1135.067,184.388,-62.259,-178.368,7.418,148.925
C06799=1135.063,184.636,-62.282,-178.365,7.420,148.924
C06800=1135.058,184.885,-62.305,-178.362,7.423,148.924
C06801=1135.053,185.133,-62.329,-178.360,7.424,148.924
C06802=1135.048,185.382,-62.352,-178.357,7.427,148.924
C06803=1135.044,185.631,-62.375,-178.354,7.430,148.924
C06804=1135.039,185.880,-62.399,-178.351,7.432,148.923
C06805=1135.034,186.129,-62.422,-178.348,7.434,148.923
C06806=1135.030,186.378,-62.445,-178.346,7.436,148.923
C06807=1135.026,186.626,-62.469,-178.343,7.439,148.923
C06808=1135.021,186.875,-62.492,-178.340,7.442,148.922
C06809=1135.017,187.125,-62.516,-178.337,7.444,148.922
C06810=1135.012,187.374,-62.539,-178.334,7.446,148.922
C06811=1135.007,187.623,-62.562,-178.331,7.449,148.922
C06812=1135.003,187.871,-62.586,-178.329,7.451,148.921
C06813=1134.998,188.120,-62.610,-178.325,7.454,148.921
C06814=1134.993,188.369,-62.633,-178.323,7.456,148.921
C06815=1134.989,188.617,-62.657,-178.320,7.458,148.921
C06816=1134.984,188.867,-62.681,-178.317,7.461,148.921
C06817=1134.980,189.116,-62.704,-178.314,7.463,148.920
C06818=1134.975,189.364,-62.728,-178.312,7.466,148.920
C06819=1134.971,189.613,-62.751,-178.309,7.469,148.920
C06820=1134.966,189.862,-62.775,-178.306,7.470,148.920
C06821=1134.961,190.110,-62.799,-178.303,7.473,148.919
C06822=1134.957,190.359,-62.822,-178.300,7.476,148.919
C06823=1134.952,190.609,-62.845,-178.298,7.478,148.919
C06824=1134.948,190.857,-62.870,-178.294,7.480,148.919
C06825=1134.943,191.106,-62.893,-178.292,7.483,148.919
C06826=1134.939,191.354,-62.917,-178.289,7.485,148.918
C06827=1134.934,191.603,-62.940,-178.286,7.488,148.918
C06828=1134.930,191.853,-62.965,-178.283,7.490,148.918
C06829=1134.925,192.102,-62.989,-178.281,7.492,148.918
C06830=1134.920,192.350,-63.013,-178.278,7.495,148.917
C06831=1134.916,192.599,-63.036,-178.274,7.498,148.917
C06832=1134.911,192.848,-63.060,-178.272,7.500,148.917
C06833=1134.906,193.097,-63.084,-178.269,7.503,148.917
C06834=1134.902,193.345,-63.108,-178.266,7.505,148.917
C06835=1134.897,193.594,-63.131,-178.263,7.507,148.916
C06836=1134.893,193.843,-63.155,-178.261,7.510,148.916
C06837=1134.887,194.092,-63.179,-178.258,7.513,148.916
C06838=1134.884,194.341,-63.203,-178.255,7.515,148.916
C06839=1134.879,194.590,-63.227,-178.252,7.518,148.915
C06840=1134.875,194.839,-63.251,-178.249,7.520,148.915
C06841=1134.870,195.087,-63.275,-178.246,7.523,148.915
C06842=1134.865,195.336,-63.299,-178.243,7.525,148.915
C06843=1134.860,195.585,-63.323,-178.241,7.528,148.915
C06844=1134.857,195.834,-63.347,-178.238,7.530,148.914
C06845=1134.852,196.083,-63.371,-178.235,7.532,148.914
C06846=1134.847,196.331,-63.395,-178.232,7.535,148.914
C06847=1134.842,196.580,-63.420,-178.229,7.538,148.914
C06848=1134.838,196.829,-63.443,-178.227,7.540,148.913
C06849=1134.833,197.077,-63.467,-178.224,7.543,148.913
C06850=1134.829,197.327,-63.491,-178.221,7.545,148.913
C06851=1134.824,197.575,-63.516,-178.218,7.548,148.913
C06852=1134.820,197.824,-63.539,-178.215,7.550,148.913
C06853=1134.815,198.073,-63.564,-178.212,7.553,148.912
C06854=1134.810,198.321,-63.588,-178.210,7.556,148.912
C06855=1134.806,198.571,-63.613,-178.206,7.558,148.912
C06856=1134.802,198.819,-63.637,-178.204,7.560,148.912
C06857=1134.797,199.068,-63.661,-178.201,7.563,148.912
C06858=1134.792,199.317,-63.685,-178.198,7.566,148.911
C06859=1134.788,199.566,-63.709,-178.196,7.568,148.911
C06860=1134.783,199.815,-63.734,-178.192,7.570,148.911
C06861=1134.779,200.063,-63.758,-178.190,7.573,148.911
C06862=1134.774,200.311,-63.782,-178.187,7.576,148.911
C06863=1134.770,200.561,-63.807,-178.184,7.578,148.910
C06864=1134.765,200.809,-63.831,-178.181,7.581,148.910
C06865=1134.761,201.058,-63.855,-178.178,7.584,148.910
C06866=1134.757,201.307,-63.880,-178.175,7.586,148.910
C06867=1134.752,201.555,-63.904,-178.173,7.588,148.910
C06868=1134.747,201.804,-63.929,-178.170,7.591,148.910
C06869=1134.743,202.053,-63.953,-178.167,7.594,148.909
C06870=1134.738,202.302,-63.978,-178.164,7.597,148.909
C06871=1134.734,202.550,-64.002,-178.162,7.599,148.909
C06872=1134.729,202.799,-64.026,-178.159,7.601,148.909
C06873=1134.725,203.048,-64.051,-178.156,7.604,148.909
C06874=1134.720,203.297,-64.075,-178.153,7.607,148.908
C06875=1134.715,203.545,-64.100,-178.150,7.609,148.908
C06876=1134.711,203.794,-64.124,-178.147,7.612,148.908
C06877=1134.706,204.043,-64.149,-178.145,7.614,148.908
C06878=1134.702,204.292,-64.173,-178.141,7.617,148.908
C06879=1134.697,204.541,-64.198,-178.139,7.619,148.907
C06880=1134.693,204.789,-64.222,-178.136,7.622,148.907
C06881=1134.689,205.038,-64.248,-178.133,7.625,148.907
C06882=1134.684,205.287,-64.273,-178.130,7.627,148.907
C06883=1134.679,205.535,-64.297,-178.127,7.630,148.907
C06884=1134.675,205.785,-64.322,-178.125,7.632,148.906
C06885=1134.670,206.033,-64.346,-178.122,7.635,148.906
C06886=1134.665,206.282,-64.371,-178.119,7.638,148.906
C06887=1134.662,206.530,-64.396,-178.116,7.641,148.906
C06888=1134.657,206.779,-64.420,-178.113,7.643,148.906
C06889=1134.652,207.029,-64.445,-178.111,7.645,148.906
C06890=1134.648,207.277,-64.470,-178.108,7.648,148.906
C06891=1134.643,207.525,-64.495,-178.105,7.651,148.905
C06892=1134.638,207.775,-64.520,-178.102,7.654,148.905
C06893=1134.634,208.023,-64.544,-178.099,7.657,148.905
C06894=1134.630,208.272,-64.570,-178.097,7.659,148.905
C06895=1134.625,208.520,-64.594,-178.093,7.661,148.905
C06896=1134.621,208.770,-64.619,-178.091,7.664,148.905
C06897=1134.616,209.040,-64.646,-178.088,7.667,148.904
C06898=1134.610,209.311,-64.673,-178.085,7.670,148.904
C06899=1134.605,209.581,-64.700,-178.082,7.672,148.904
C06900=1134.601,209.851,-64.728,-178.078,7.676,148.904
C06901=1134.596,210.101,-64.753,-178.076,7.678,148.904
C06902=1134.591,210.350,-64.777,-178.073,7.681,148.903
C06903=1134.588,210.598,-64.803,-178.070,7.684,148.903
C06904=1134.583,210.847,-64.827,-178.067,7.686,148.903
C06905=1134.578,211.096,-64.853,-178.064,7.689,148.903
C06906=1134.574,211.344,-64.877,-178.062,7.691,148.903
C06907=1134.570,211.593,-64.903,-178.059,7.694,148.903
C06908=1134.565,211.842,-64.928,-178.056,7.697,148.902
C06909=1134.560,212.090,-64.953,-178.053,7.700,148.902
C06910=1134.555,212.339,-64.978,-178.050,7.702,148.902
C06911=1134.552,212.588,-65.003,-178.047,7.705,148.902
C06912=1134.547,212.836,-65.028,-178.045,7.707,148.902
C06913=1134.542,213.085,-65.054,-178.042,7.710,148.902
C06914=1134.538,213.333,-65.079,-178.039,7.713,148.902
C06915=1134.533,213.583,-65.104,-178.036,7.716,148.901
C06916=1134.528,213.831,-65.129,-178.033,7.719,148.901
C06917=1134.524,214.080,-65.154,-178.030,7.721,148.901
C06918=1134.520,214.329,-65.180,-178.027,7.724,148.901
C06919=1134.515,214.577,-65.205,-178.025,7.726,148.901
C06920=1134.511,214.826,-65.230,-178.022,7.729,148.901
C06921=1134.506,215.074,-65.255,-178.019,7.732,148.901
C06922=1134.502,215.323,-65.281,-178.016,7.735,148.900
C06923=1134.497,215.571,-65.306,-178.013,7.737,148.900
C06924=1134.492,215.821,-65.332,-178.010,7.740,148.900
C06925=1134.489,216.069,-65.357,-178.008,7.743,148.900
C06926=1134.484,216.317,-65.382,-178.005,7.745,148.900
C06927=1134.480,216.567,-65.407,-178.002,7.748,148.900
C06928=1134.475,216.815,-65.433,-177.999,7.751,148.899
C06929=1134.471,217.063,-65.458,-177.996,7.754,148.899
C06930=1134.466,217.312,-65.484,-177.994,7.757,148.899
C06931=1134.462,217.561,-65.510,-177.991,7.759,148.899
C06932=1134.457,217.809,-65.535,-177.988,7.762,148.899
C06933=1134.453,218.059,-65.560,-177.985,7.765,148.899
C06934=1134.448,218.307,-65.586,-177.983,7.767,148.899
C06935=1134.444,218.556,-65.611,-177.980,7.770,148.898
C06936=1134.440,218.804,-65.637,-177.977,7.773,148.898
C06937=1134.435,219.052,-65.662,-177.974,7.776,148.898
C06938=1134.430,219.301,-65.688,-177.971,7.779,148.898
C06939=1134.426,219.550,-65.714,-177.968,7.781,148.898
C06940=1134.422,219.799,-65.740,-177.965,7.784,148.898
C06941=1134.417,220.047,-65.765,-177.962,7.787,148.898
C06942=1134.413,220.296,-65.791,-177.960,7.790,148.898
C06943=1134.409,220.545,-65.817,-177.957,7.792,148.897
C06944=1134.403,220.793,-65.843,-177.955,7.795,148.897
C06945=1134.381,222.054,-65.973,-178.885,9.564,149.580
C06946=1134.377,222.303,-65.998,-178.883,9.568,149.580
C06947=1134.373,222.552,-66.024,-178.880,9.571,149.580
C06948=1134.367,222.799,-66.051,-178.876,9.574,149.580
C06949=1134.363,223.048,-66.077,-178.874,9.577,149.580
C06950=1134.359,223.297,-66.102,-178.871,9.581,149.580
C06951=1134.354,223.546,-66.129,-178.868,9.584,149.580
C06952=1134.350,223.794,-66.155,-178.865,9.588,149.580
C06953=1134.346,224.043,-66.181,-178.861,9.592,149.580
C06954=1134.341,224.292,-66.208,-178.859,9.594,149.580
C06955=1134.336,224.540,-66.233,-178.855,9.598,149.580
C06956=1134.332,224.788,-66.260,-178.852,9.602,149.580
C06957=1134.327,225.037,-66.286,-178.849,9.605,149.580
C06958=1134.323,225.275,-66.312,-178.846,9.608,149.580
C06959=1134.320,225.511,-66.336,-178.843,9.611,149.580
C06960=1134.315,225.748,-66.361,-178.839,9.615,149.579
C06961=1134.311,225.984,-66.386,-178.836,9.619,149.580
C06962=1134.307,226.222,-66.412,-178.833,9.621,149.579
C06963=1134.302,226.459,-66.437,-178.829,9.625,149.579
C06964=1134.298,226.695,-66.462,-178.826,9.628,149.579
C06965=1134.294,226.933,-66.487,-178.822,9.632,149.579
C06966=1134.290,227.181,-66.514,-178.819,9.635,149.579
C06967=1134.285,227.430,-66.540,-178.815,9.639,149.579
C06968=1134.281,227.678,-66.567,-178.812,9.642,149.579
C06969=1134.276,227.927,-66.594,-178.808,9.646,149.579
C06970=1134.272,228.176,-66.619,-178.804,9.649,149.578
C06971=1134.268,228.424,-66.647,-178.801,9.653,149.578
C06972=1134.264,228.672,-66.673,-178.797,9.656,149.578
C06973=1134.259,228.921,-66.699,-178.793,9.661,149.578
C06974=1134.255,229.170,-66.726,-178.789,9.664,149.578
C06975=1134.250,229.418,-66.753,-178.785,9.667,149.578
C06976=1134.246,229.666,-66.779,-178.781,9.671,149.577
C06977=1134.241,229.915,-66.806,-178.777,9.675,149.577
C06978=1134.237,230.164,-66.833,-178.773,9.678,149.577
C06979=1134.233,230.412,-66.859,-178.769,9.682,149.577
C06980=1134.228,230.661,-66.886,-178.765,9.686,149.577
C06981=1134.223,230.909,-66.913,-178.761,9.689,149.576
C06982=1134.219,231.157,-66.940,-178.758,9.693,149.576
C06983=1134.214,231.406,-66.966,-178.754,9.696,149.576
C06984=1134.210,231.655,-66.993,-178.750,9.699,149.576
C06985=1134.206,231.903,-67.020,-178.747,9.703,149.576
C06986=1134.201,232.152,-67.047,-178.743,9.705,149.575
C06987=1134.197,232.400,-67.074,-178.740,9.709,149.575
C06988=1134.193,232.649,-67.101,-178.736,9.712,149.575
C06989=1134.189,232.897,-67.128,-178.733,9.716,149.575
C06990=1134.184,233.146,-67.155,-178.729,9.718,149.575
C06991=1134.179,233.394,-67.182,-178.726,9.722,149.575
C06992=1134.175,233.643,-67.208,-178.723,9.724,149.575
C06993=1134.171,233.891,-67.235,-178.719,9.728,149.574
C06994=1134.166,234.140,-67.262,-178.716,9.731,149.574
C06995=1134.162,234.389,-67.290,-178.713,9.733,149.574
C06996=1134.158,234.637,-67.318,-178.709,9.737,149.574
C06997=1134.154,234.885,-67.344,-178.706,9.739,149.574
C06998=1134.149,235.133,-67.371,-178.703,9.742,149.574
C06999=1134.144,235.382,-67.398,-178.700,9.745,149.573
C07000=1134.140,235.630,-67.425,-178.697,9.748,149.573
C07001=1134.136,235.880,-67.453,-178.694,9.750,149.573
C07002=1134.131,236.128,-67.480,-178.691,9.753,149.573
C07003=1134.127,236.376,-67.507,-178.689,9.756,149.573
C07004=1134.123,236.624,-67.534,-178.686,9.759,149.573
C07005=1134.119,236.873,-67.561,-178.683,9.762,149.573
C07006=1134.114,237.122,-67.588,-178.680,9.764,149.573
C07007=1134.110,237.370,-67.616,-178.677,9.767,149.573
C07008=1134.105,237.618,-67.643,-178.675,9.769,149.573
C07009=1134.100,237.867,-67.670,-178.672,9.772,149.572
C07010=1134.096,238.116,-67.698,-178.669,9.775,149.572
C07011=1134.092,238.364,-67.726,-178.667,9.777,149.572
C07012=1134.087,238.612,-67.753,-178.664,9.780,149.572
C07013=1134.083,238.861,-67.780,-178.662,9.782,149.572
C07014=1134.079,239.074,-67.804,-178.660,9.784,149.572
C07015=1134.076,239.289,-67.827,-178.658,9.786,149.572
C07016=1134.072,239.503,-67.850,-178.656,9.788,149.572
C07017=1134.069,239.717,-67.874,-178.654,9.791,149.572
C07018=1134.065,239.932,-67.898,-178.651,9.793,149.572
C07019=1134.061,240.146,-67.921,-178.650,9.794,149.572
C07020=1134.057,240.360,-67.945,-178.648,9.796,149.572
C07021=1134.053,240.574,-67.968,-178.646,9.798,149.572
C07022=1134.049,240.823,-67.997,-178.644,9.801,149.572
C07023=1134.045,241.071,-68.024,-178.642,9.803,149.572
C07024=1134.040,241.319,-68.051,-178.640,9.805,149.572
C07025=1134.036,241.568,-68.079,-178.638,9.807,149.572
C07026=1134.032,241.817,-68.106,-178.636,9.810,149.572
C07027=1134.027,242.064,-68.134,-178.634,9.812,149.572
C07028=1134.023,242.313,-68.161,-178.632,9.814,149.572
C07029=1134.018,242.562,-68.190,-178.631,9.816,149.572
C07030=1134.014,242.810,-68.217,-178.629,9.818,149.572
C07031=1134.009,243.058,-68.244,-178.627,9.821,149.572
C07032=1134.005,243.307,-68.272,-178.625,9.823,149.572
C07033=1134.001,243.555,-68.300,-178.624,9.824,149.572
C07034=1133.996,243.804,-68.327,-178.622,9.827,149.572
C07035=1133.992,244.052,-68.355,-178.621,9.829,149.573
C07036=1133.988,244.301,-68.382,-178.619,9.831,149.573
C07037=1133.984,244.549,-68.410,-178.618,9.833,149.573
C07038=1133.980,244.797,-68.438,-178.617,9.835,149.573
C07039=1133.975,245.046,-68.465,-178.615,9.837,149.573
C07040=1133.971,245.294,-68.493,-178.615,9.839,149.573
C07041=1133.966,245.543,-68.521,-178.613,9.841,149.573
C07042=1133.961,245.791,-68.548,-178.612,9.843,149.574
C07043=1133.958,246.040,-68.577,-178.611,9.845,149.574
C07044=1133.953,246.288,-68.604,-178.610,9.847,149.574
C07045=1133.949,246.536,-68.631,-178.608,9.849,149.574
C07046=1133.945,246.785,-68.659,-178.607,9.851,149.574
C07047=1133.940,247.033,-68.687,-178.607,9.853,149.575
C07048=1133.936,247.282,-68.715,-178.606,9.855,149.575
C07049=1133.931,247.530,-68.742,-178.601,9.859,149.574
C07050=1133.927,247.778,-68.770,-178.593,9.865,149.574
C07051=1133.923,248.027,-68.798,-178.585,9.871,149.573
C07052=1133.918,248.275,-68.825,-178.577,9.877,149.572
C07053=1133.914,248.524,-68.854,-178.570,9.882,149.572
C07054=1133.910,248.772,-68.882,-178.563,9.887,149.571
C07055=1133.905,249.020,-68.910,-178.556,9.893,149.571
C07056=1133.901,249.269,-68.938,-178.550,9.897,149.570
C07057=1133.896,249.517,-68.965,-178.543,9.902,149.570
C07058=1133.892,249.766,-68.994,-178.538,9.906,149.569
C07059=1133.888,250.014,-69.021,-178.532,9.911,149.569
C07060=1133.884,250.263,-69.050,-178.527,9.914,149.568
C07061=1133.880,250.511,-69.078,-178.522,9.918,149.568
C07062=1133.875,250.760,-69.107,-178.517,9.922,149.567
C07063=1133.871,251.008,-69.135,-178.513,9.926,149.567
C07064=1133.867,251.256,-69.163,-178.509,9.929,149.567
C07065=1133.862,251.505,-69.191,-178.505,9.931,149.567
C07066=1133.858,251.752,-69.220,-178.501,9.934,149.566
C07067=1133.854,252.001,-69.249,-178.498,9.937,149.566
C07068=1133.849,252.249,-69.276,-178.495,9.939,149.566
C07069=1133.845,252.498,-69.305,-178.493,9.941,149.566
C07070=1133.842,252.712,-69.329,-178.491,9.943,149.566
C07071=1133.838,252.926,-69.353,-178.489,9.945,149.566
C07072=1133.834,253.140,-69.378,-178.487,9.947,149.565
C07073=1133.830,253.354,-69.402,-178.486,9.949,149.565
C07074=1133.827,253.568,-69.427,-178.485,9.949,149.566
C07075=1133.823,253.782,-69.452,-178.484,9.951,149.566
C07076=1133.819,253.997,-69.476,-178.483,9.952,149.566
C07077=1133.815,254.211,-69.501,-178.483,9.953,149.566
C07078=1133.811,254.458,-69.529,-178.483,9.954,149.566
C07079=1133.807,254.707,-69.558,-178.483,9.955,149.566
C07080=1133.803,254.955,-69.586,-178.483,9.955,149.566
C07081=1133.798,255.203,-69.614,-178.484,9.956,149.567
C07082=1133.794,255.452,-69.642,-178.485,9.957,149.567
C07083=1133.789,255.700,-69.671,-178.486,9.957,149.568
C07084=1133.785,255.948,-69.700,-178.487,9.957,149.568
C07085=1133.781,256.197,-69.728,-178.484,9.960,149.568
C07086=1133.777,256.445,-69.756,-178.481,9.963,149.568
C07087=1133.772,256.694,-69.785,-178.478,9.966,149.568
C07088=1133.768,256.942,-69.813,-178.476,9.969,149.568
C07089=1133.764,257.190,-69.842,-178.473,9.972,149.568
C07090=1133.760,257.439,-69.870,-178.470,9.974,149.568
C07091=1133.755,257.687,-69.899,-178.466,9.978,149.567
C07092=1133.750,257.936,-69.927,-178.463,9.981,149.567
C07093=1133.747,258.184,-69.956,-178.460,9.983,149.567
C07094=1133.742,258.432,-69.985,-178.457,9.987,149.567
C07095=1133.738,258.680,-70.013,-178.454,9.990,149.567
C07096=1133.734,258.929,-70.042,-178.450,9.992,149.567
C07097=1133.729,259.176,-70.070,-178.447,9.996,149.567
C07098=1133.725,259.425,-70.099,-178.444,9.998,149.566
C07099=1133.721,259.674,-70.128,-178.440,10.002,149.566
C07100=1133.716,259.922,-70.156,-178.437,10.005,149.566
C07101=1133.712,260.170,-70.185,-178.433,10.008,149.566
C07102=1133.708,260.419,-70.214,-178.430,10.011,149.566
C07103=1133.704,260.666,-70.243,-178.426,10.014,149.566
C07104=1133.699,260.915,-70.271,-178.423,10.017,149.566
C07105=1133.695,261.163,-70.301,-178.419,10.020,149.565
C07106=1133.691,261.412,-70.329,-178.415,10.024,149.565
C07107=1133.686,261.659,-70.358,-178.412,10.026,149.565
C07108=1133.682,261.908,-70.387,-178.408,10.030,149.565
C07109=1133.678,262.156,-70.416,-178.404,10.033,149.564
C07110=1133.674,262.405,-70.444,-178.400,10.036,149.564
C07111=1133.669,262.653,-70.473,-178.397,10.040,149.564
C07112=1133.665,262.901,-70.502,-178.393,10.043,149.564
C07113=1133.661,263.150,-70.532,-178.389,10.046,149.564
C07114=1133.656,263.398,-70.561,-178.385,10.049,149.563
C07115=1133.652,263.646,-70.589,-178.381,10.053,149.563
C07116=1133.648,263.894,-70.618,-178.377,10.056,149.563
C07117=1133.644,264.142,-70.648,-178.373,10.059,149.562
C07118=1133.639,264.391,-70.677,-178.369,10.062,149.562
C07119=1133.635,264.640,-70.706,-178.366,10.065,149.562
C07120=1133.631,264.888,-70.735,-178.364,10.067,149.562
C07121=1133.626,265.135,-70.765,-178.362,10.069,149.562
C07122=1133.622,265.384,-70.793,-178.359,10.072,149.562
C07123=1133.618,265.632,-70.822,-178.356,10.074,149.562
C07124=1133.614,265.880,-70.852,-178.354,10.076,149.562
C07125=1133.610,266.129,-70.881,-178.351,10.079,149.561
C07126=1133.606,266.343,-70.906,-178.349,10.081,149.562
C07127=1133.602,266.557,-70.931,-178.348,10.082,149.561
C07128=1133.599,266.771,-70.957,-178.345,10.084,149.561
C07129=1133.595,266.985,-70.981,-178.343,10.086,149.561
C07130=1133.591,267.198,-71.006,-178.341,10.088,149.561
C07131=1133.587,267.412,-71.032,-178.339,10.090,149.561
C07132=1133.584,267.627,-71.057,-178.336,10.092,149.561
C07133=1133.580,267.840,-71.082,-178.335,10.095,149.561
C07134=1133.576,268.088,-71.112,-178.332,10.097,149.561
C07135=1133.572,268.337,-71.141,-178.329,10.099,149.561
C07136=1133.568,268.585,-71.171,-178.326,10.102,149.561
C07137=1133.563,268.833,-71.200,-178.323,10.105,149.561
C07138=1133.559,269.081,-71.230,-178.321,10.107,149.560
C07139=1133.554,269.329,-71.259,-178.318,10.110,149.560
C07140=1133.550,269.577,-71.288,-178.315,10.112,149.560
C07141=1133.546,269.825,-71.318,-178.313,10.114,149.560
C07142=1133.542,270.074,-71.346,-178.310,10.117,149.560
C07143=1133.538,270.322,-71.376,-178.307,10.120,149.560
C07144=1133.533,270.570,-71.406,-178.305,10.122,149.560
C07145=1133.529,270.819,-71.435,-178.302,10.125,149.560
C07146=1133.525,271.067,-71.465,-178.299,10.127,149.560
C07147=1133.521,271.315,-71.494,-178.296,10.130,149.559
C07148=1133.516,271.564,-71.524,-178.293,10.133,149.559
C07149=1133.512,271.812,-71.554,-178.290,10.136,149.559
C07150=1133.508,272.060,-71.583,-178.288,10.138,149.559
C07151=1133.503,272.308,-71.613,-178.285,10.140,149.559
C07152=1133.499,272.557,-71.642,-178.282,10.143,149.559
C07153=1133.495,272.805,-71.672,-178.279,10.146,149.559
C07154=1133.491,273.053,-71.701,-178.276,10.149,149.559
C07155=1133.487,273.301,-71.731,-178.273,10.151,149.558
C07156=1133.483,273.549,-71.761,-178.270,10.154,149.558
C07157=1133.478,273.798,-71.791,-178.267,10.157,149.558
C07158=1133.474,274.046,-71.820,-178.264,10.159,149.558
C07159=1133.470,274.294,-71.850,-178.261,10.162,149.558
C07160=1133.466,274.542,-71.880,-178.258,10.165,149.558
C07161=1133.462,274.790,-71.909,-178.254,10.168,149.558
C07162=1133.457,275.038,-71.939,-178.251,10.171,149.558
C07163=1133.452,275.287,-71.969,-178.248,10.173,149.557
C07164=1133.449,275.535,-71.999,-178.245,10.176,149.557
C07165=1133.444,275.783,-72.028,-178.242,10.179,149.557
C07166=1133.440,276.031,-72.058,-178.238,10.181,149.557
C07167=1133.436,276.279,-72.089,-178.235,10.185,149.557
C07168=1133.431,276.527,-72.118,-178.232,10.188,149.557
C07169=1133.427,276.776,-72.147,-178.229,10.190,149.556
C07170=1133.423,277.023,-72.178,-178.226,10.193,149.556
C07171=1133.418,277.272,-72.208,-178.222,10.196,149.556
C07172=1133.415,277.520,-72.238,-178.219,10.199,149.556
C07173=1133.411,277.769,-72.268,-178.215,10.201,149.556
C07174=1133.407,278.016,-72.298,-178.212,10.205,149.556
C07175=1133.402,278.265,-72.328,-178.209,10.207,149.555
C07176=1133.398,278.512,-72.358,-178.205,10.209,149.555
C07177=1133.394,278.761,-72.388,-178.202,10.213,149.555
C07178=1133.389,279.009,-72.418,-178.198,10.215,149.555
C07179=1133.385,279.257,-72.448,-178.195,10.219,149.555
C07180=1133.381,279.505,-72.478,-178.191,10.221,149.554
C07181=1133.377,279.754,-72.508,-178.187,10.224,149.554
C07182=1133.373,279.968,-72.534,-178.184,10.227,149.554
C07183=1133.370,280.181,-72.560,-178.181,10.230,149.554
C07184=1133.366,280.395,-72.586,-178.179,10.232,149.553
C07185=1133.362,280.609,-72.612,-178.175,10.234,149.553
C07186=1133.359,280.822,-72.638,-178.172,10.236,149.553
C07187=1133.355,281.037,-72.664,-178.169,10.239,149.553
C07188=1133.351,281.250,-72.691,-178.166,10.242,149.552
C07189=1133.348,281.464,-72.716,-178.163,10.244,149.552
C07190=1133.344,281.712,-72.747,-178.159,10.247,149.552
C07191=1133.339,281.960,-72.777,-178.157,10.250,149.552
C07192=1133.335,282.209,-72.808,-178.153,10.252,149.552
C07193=1133.332,282.456,-72.838,-178.150,10.255,149.552
C07194=1133.327,282.704,-72.869,-178.147,10.257,149.552
C07195=1133.323,282.953,-72.898,-178.144,10.260,149.551
C07196=1133.318,283.200,-72.929,-178.141,10.263,149.551
C07197=1133.315,283.449,-72.959,-178.138,10.264,149.551
C07198=1133.310,283.697,-72.990,-178.135,10.267,149.551
C07199=1133.306,283.945,-73.020,-178.132,10.269,149.550
C07200=1133.301,284.193,-73.050,-178.129,10.272,149.550
C07201=1133.297,284.442,-73.082,-178.126,10.275,149.550
C07202=1133.294,284.689,-73.112,-178.123,10.277,149.550
C07203=1133.289,284.937,-73.142,-178.120,10.280,149.550
C07204=1133.285,285.185,-73.173,-178.117,10.283,149.550
C07205=1133.281,285.434,-73.204,-178.114,10.285,149.550
C07206=1133.276,285.682,-73.235,-178.110,10.288,149.549
C07207=1133.272,285.930,-73.264,-178.107,10.291,149.549
C07208=1133.268,286.178,-73.295,-178.105,10.292,149.549
C07209=1133.264,286.426,-73.325,-178.102,10.295,149.549
C07210=1133.260,286.674,-73.356,-178.099,10.298,149.549
C07211=1133.255,286.922,-73.387,-178.095,10.300,149.548
C07212=1133.252,287.170,-73.417,-178.092,10.303,149.548
C07213=1133.247,287.418,-73.448,-178.089,10.305,149.548
C07214=1133.243,287.666,-73.479,-178.086,10.308,149.548
C07215=1133.239,287.915,-73.509,-178.083,10.310,149.548
C07216=1133.235,288.163,-73.540,-178.080,10.313,149.548
C07217=1133.230,288.411,-73.571,-178.077,10.316,149.547
C07218=1133.227,288.659,-73.601,-178.074,10.318,149.547
C07219=1133.223,288.906,-73.633,-178.071,10.320,149.547
C07220=1133.218,289.154,-73.664,-178.068,10.323,149.547
C07221=1133.214,289.403,-73.695,-178.065,10.326,149.547
C07222=1133.210,289.651,-73.725,-178.062,10.328,149.546
C07223=1133.206,289.899,-73.756,-178.059,10.331,149.546
C07224=1133.201,290.147,-73.787,-178.055,10.333,149.546
C07225=1133.197,290.395,-73.818,-178.053,10.336,149.546
C07226=1133.194,290.643,-73.849,-178.049,10.338,149.546
C07227=1133.189,290.891,-73.880,-178.046,10.341,149.546
C07228=1133.185,291.139,-73.910,-178.043,10.344,149.545
C07229=1133.181,291.387,-73.942,-178.040,10.346,149.545
C07230=1133.176,291.635,-73.972,-178.037,10.349,149.545
C07231=1133.173,291.883,-74.004,-178.034,10.351,149.545
C07232=1133.168,292.131,-74.034,-178.031,10.353,149.545
C07233=1133.164,292.380,-74.065,-178.028,10.356,149.544
C07234=1133.160,292.627,-74.097,-178.025,10.358,149.544
C07235=1133.155,292.875,-74.128,-178.022,10.361,149.544
C07236=1133.151,293.124,-74.159,-178.019,10.364,149.544
C07237=1133.147,293.371,-74.190,-178.015,10.366,149.544
C07238=1133.144,293.585,-74.217,-178.013,10.368,149.544
C07239=1133.140,293.799,-74.244,-178.010,10.371,149.544
C07240=1133.137,294.012,-74.271,-178.008,10.373,149.543
C07241=1133.133,294.226,-74.297,-178.005,10.375,149.543
C07242=1133.130,294.439,-74.324,-178.002,10.377,149.543
C07243=1133.126,294.653,-74.351,-178.000,10.379,149.543
C07244=1133.123,294.867,-74.378,-177.997,10.382,149.543
C07245=1133.119,295.081,-74.405,-177.994,10.384,149.543
C07246=1133.115,295.329,-74.436,-177.991,10.386,149.542
C07247=1133.111,295.577,-74.467,-177.988,10.389,149.542
C07248=1133.106,295.825,-74.498,-177.985,10.391,149.542
C07249=1133.103,296.073,-74.530,-177.982,10.394,149.542
C07250=1133.098,296.321,-74.561,-177.978,10.397,149.542
C07251=1133.094,296.569,-74.593,-177.976,10.399,149.541
C07252=1133.090,296.817,-74.623,-177.972,10.402,149.541
C07253=1133.086,297.065,-74.655,-177.970,10.404,149.541
C07254=1133.082,297.312,-74.687,-177.967,10.406,149.541
C07255=1133.078,297.561,-74.718,-177.964,10.409,149.541
C07256=1133.073,297.808,-74.749,-177.960,10.411,149.540
C07257=1133.069,298.057,-74.780,-177.957,10.414,149.540
C07258=1133.065,298.304,-74.812,-177.954,10.417,149.540
C07259=1133.061,298.552,-74.844,-177.951,10.419,149.540
C07260=1133.057,298.800,-74.875,-177.948,10.422,149.540
C07261=1133.053,299.048,-74.906,-177.945,10.425,149.540
C07262=1133.049,299.296,-74.938,-177.942,10.427,149.539
C07263=1133.045,299.544,-74.969,-177.939,10.430,149.539
C07264=1133.040,299.793,-75.001,-177.935,10.432,149.539
C07265=1133.036,300.040,-75.033,-177.932,10.435,149.539
C07266=1133.032,300.289,-75.064,-177.929,10.437,149.539
C07267=1133.028,300.537,-75.096,-177.927,10.439,149.539
C07268=1133.024,300.784,-75.127,-177.923,10.442,149.538
C07269=1133.020,301.032,-75.159,-177.920,10.445,149.538
C07270=1133.016,301.280,-75.190,-177.917,10.447,149.538
C07271=1133.011,301.528,-75.222,-177.914,10.450,149.538
C07272=1133.008,301.776,-75.254,-177.911,10.452,149.538
C07273=1133.003,302.024,-75.286,-177.908,10.455,149.538
C07274=1133.000,302.272,-75.318,-177.905,10.457,149.537
C07275=1132.995,302.520,-75.350,-177.901,10.460,149.537
C07276=1132.991,302.768,-75.381,-177.898,10.463,149.537
C07277=1132.987,303.016,-75.413,-177.895,10.465,149.537
C07278=1132.982,303.263,-75.444,-177.892,10.468,149.537
C07279=1132.979,303.511,-75.476,-177.889,10.470,149.536
C07280=1132.974,303.760,-75.508,-177.886,10.473,149.536
C07281=1132.970,304.007,-75.540,-177.882,10.475,149.536
C07282=1132.966,304.255,-75.572,-177.879,10.478,149.536
C07283=1132.962,304.503,-75.604,-177.877,10.480,149.536
C07284=1132.958,304.752,-75.636,-177.874,10.483,149.536
C07285=1132.954,304.999,-75.668,-177.871,10.485,149.535
C07286=1132.949,305.247,-75.700,-177.867,10.487,149.535
C07287=1132.946,305.495,-75.732,-177.864,10.490,149.535
C07288=1132.941,305.743,-75.763,-177.861,10.493,149.535
C07289=1132.937,305.991,-75.796,-177.858,10.495,149.535
C07290=1132.933,306.239,-75.828,-177.855,10.498,149.534
C07291=1132.929,306.486,-75.859,-177.852,10.501,149.534
C07292=1132.925,306.735,-75.891,-177.848,10.503,149.534
C07293=1132.921,306.983,-75.923,-177.845,10.506,149.534
C07294=1132.918,307.196,-75.951,-177.843,10.508,149.534
C07295=1132.914,307.409,-75.979,-177.840,10.510,149.534
C07296=1132.911,307.623,-76.007,-177.838,10.512,149.533
C07297=1132.907,307.837,-76.034,-177.835,10.514,149.533
C07298=1132.904,308.050,-76.062,-177.832,10.517,149.533
C07299=1132.900,308.263,-76.090,-177.830,10.519,149.533
C07300=1132.897,308.477,-76.117,-177.826,10.521,149.533
C07301=1132.893,308.691,-76.145,-177.824,10.523,149.533
C07302=1132.889,308.938,-76.177,-177.821,10.526,149.532
C07303=1132.884,309.186,-76.209,-177.818,10.528,149.532
C07304=1132.880,309.434,-76.241,-177.814,10.531,149.532
C07305=1132.876,309.682,-76.274,-177.811,10.533,149.532
C07306=1132.873,309.930,-76.306,-177.808,10.536,149.532
C07307=1132.868,310.178,-76.339,-177.805,10.538,149.531
C07308=1132.864,310.425,-76.370,-177.802,10.541,149.531
C07309=1132.860,310.673,-76.403,-177.799,10.544,149.531
